LIN {X 0,Y 477.289,Z 363.649,A -85,B 0,C 180,E1 -7445.274,E2 -7445.274} C_VEL
LIN {X 0,Y 471.666,Z 382.664,A -85,B 0,C 180,E1 -7445.357,E2 -7445.357} C_VEL
LIN {X 0,Y 470.971,Z 388.509,A -85,B 0,C 180,E1 -7445.422,E2 -7445.422} C_VEL
LIN {X 0,Y 470.744,Z 411.297,A -85,B 0,C 180,E1 -7445.812,E2 -7445.812} C_VEL
LIN {X 0,Y 470.533,Z 424.379,A -85,B 0,C 180,E1 -7446.217,E2 -7446.217} C_VEL
LIN {X 0,Y 470.087,Z 436.738,A -85,B 0,C 180,E1 -7446.777,E2 -7446.777} C_VEL
LIN {X 0,Y 469.665,Z 447.889,A -85,B 0,C 180,E1 -7447.453,E2 -7447.453} C_VEL
LIN {X 0,Y 469.142,Z 459.604,A -85,B 0,C 180,E1 -7448.361,E2 -7448.361} C_VEL
LIN {X 0,Y 468.636,Z 469.87,A -85,B 0,C 180,E1 -7449.365,E2 -7449.365} C_VEL
LIN {X 0,Y 468.188,Z 479.141,A -85,B 0,C 180,E1 -7450.489,E2 -7450.489} C_VEL
LIN {X 0,Y 467.745,Z 486.733,A -85,B 0,C 180,E1 -7451.608,E2 -7451.608} C_VEL
LIN {X 0,Y 467.41,Z 494.144,A -85,B 0,C 180,E1 -7452.951,E2 -7452.951} C_VEL
LIN {X 0,Y 467.098,Z 500.27,A -85,B 0,C 180,E1 -7454.357,E2 -7454.357} C_VEL
LIN {X 0,Y 466.929,Z 504.578,A -85,B 0,C 180,E1 -7455.621,E2 -7455.621} C_VEL
LIN {X 0,Y 466.792,Z 508.016,A -85,B 0,C 180,E1 -7456.948,E2 -7456.948} C_VEL
LIN {X 0,Y 466.745,Z 510.263,A -85,B 0,C 180,E1 -7458.166,E2 -7458.166} C_VEL
LIN {X 0,Y 466.637,Z 511.87,A -85,B 0,C 180,E1 -7459.588,E2 -7459.588} C_VEL
LIN {X 0,Y 466.582,Z 512.309,A -85,B 0,C 180,E1 -7460.463,E2 -7460.463} C_VEL
LIN {X 0,Y 466.636,Z 512.343,A -85,B 0,C 180,E1 -7461.338,E2 -7461.338} C_VEL
LIN {X 0,Y 466.705,Z 511.259,A -85,B 0,C 180,E1 -7463.081,E2 -7463.081} C_VEL
LIN {X 0,Y 466.765,Z 510.083,A -85,B 0,C 180,E1 -7463.95,E2 -7463.95} C_VEL
LIN {X 0,Y 466.742,Z 508.508,A -85,B 0,C 180,E1 -7464.817,E2 -7464.817} C_VEL
LIN {X 0,Y 466.893,Z 505.337,A -85,B 0,C 180,E1 -7466.117,E2 -7466.117} C_VEL
LIN {X 0,Y 466.996,Z 501.127,A -85,B 0,C 180,E1 -7467.413,E2 -7467.413} C_VEL
LIN {X 0,Y 467.29,Z 494.749,A -85,B 0,C 180,E1 -7468.923,E2 -7468.923} C_VEL
LIN {X 0,Y 467.608,Z 487.78,A -85,B 0,C 180,E1 -7470.216,E2 -7470.216} C_VEL
LIN {X 0,Y 468.041,Z 479.089,A -85,B 0,C 180,E1 -7471.506,E2 -7471.506} C_VEL
LIN {X 0,Y 468.446,Z 469.254,A -85,B 0,C 180,E1 -7472.688,E2 -7472.688} C_VEL
LIN {X 0,Y 468.883,Z 459.22,A -85,B 0,C 180,E1 -7473.653,E2 -7473.653} C_VEL
LIN {X 0,Y 469.362,Z 448.098,A -85,B 0,C 180,E1 -7474.509,E2 -7474.509} C_VEL
LIN {X 0,Y 469.775,Z 437.576,A -85,B 0,C 180,E1 -7475.15,E2 -7475.15} C_VEL
LIN {X 0,Y 470.065,Z 424.945,A -85,B 0,C 180,E1 -7475.739,E2 -7475.739} C_VEL
LIN {X 0,Y 470.376,Z 412.214,A -85,B 0,C 180,E1 -7476.139,E2 -7476.139} C_VEL
LIN {X 0,Y 470.57,Z 394.34,A -85,B 0,C 180,E1 -7476.459,E2 -7476.459} C_VEL
LIN {X 0,Y 471.157,Z 315.376,A -85,B 0,C 180,E1 -7477.664,E2 -7477.664} C_VEL
LIN {X 0,Y 468.446,Z 301.546,A -85,B 0,C 180,E1 -7478,E2 -7478} C_VEL
LIN {X 0,Y 468.444,Z 292.876,A -85,B 0,C 180,E1 -7479.718,E2 -7479.718} C_VEL
LIN {X 0,Y 467.617,Z 287.24,A -85,B 0,C 180,E1 -7480.911,E2 -7480.911} C_VEL
LIN {X 0,Y 467.59,Z 287.239,A -85,B 0,C 180,E1 -7483.03,E2 -7483.03} C_VEL
LIN {X 0,Y 467.655,Z 287.227,A -85,B 0,C 180,E1 -7485.885,E2 -7485.885} C_VEL
LIN {X 0,Y 467.623,Z 287.232,A -85,B 0,C 180,E1 -7489.308,E2 -7489.308} C_VEL
LIN {X 0,Y 467.537,Z 287.242,A -85,B 0,C 180,E1 -7492.074,E2 -7492.074} C_VEL
LIN {X 0,Y 467.561,Z 287.247,A -85,B 0,C 180,E1 -7494.89,E2 -7494.89} C_VEL
LIN {X 0,Y 467.549,Z 287.24,A -85,B 0,C 180,E1 -7497.774,E2 -7497.774} C_VEL
LIN {X 0,Y 467.548,Z 287.248,A -85,B 0,C 180,E1 -7501.04,E2 -7501.04} C_VEL
LIN {X 0,Y 467.582,Z 287.236,A -85,B 0,C 180,E1 -7504.24,E2 -7504.24} C_VEL
LIN {X 0,Y 467.548,Z 287.248,A -85,B 0,C 180,E1 -7507.185,E2 -7507.185} C_VEL
LIN {X 0,Y 467.562,Z 287.238,A -85,B 0,C 180,E1 -7510.267,E2 -7510.267} C_VEL
LIN {X 0,Y 467.55,Z 287.242,A -85,B 0,C 180,E1 -7513.746,E2 -7513.746} C_VEL
LIN {X 0,Y 467.549,Z 287.24,A -85,B 0,C 180,E1 -7516.254,E2 -7516.254} C_VEL
LIN {X 0,Y 467.561,Z 287.242,A -85,B 0,C 180,E1 -7519.733,E2 -7519.733} C_VEL
LIN {X 0,Y 467.527,Z 287.243,A -85,B 0,C 180,E1 -7522.818,E2 -7522.818} C_VEL
LIN {X 0,Y 467.581,Z 287.241,A -85,B 0,C 180,E1 -7525.76,E2 -7525.76} C_VEL
LIN {X 0,Y 467.572,Z 287.238,A -85,B 0,C 180,E1 -7528.955,E2 -7528.955} C_VEL
LIN {X 0,Y 467.608,Z 287.233,A -85,B 0,C 180,E1 -7532.469,E2 -7532.469} C_VEL
LIN {X 0,Y 467.559,Z 287.24,A -85,B 0,C 180,E1 -7535.11,E2 -7535.11} C_VEL
LIN {X 0,Y 467.539,Z 287.248,A -85,B 0,C 180,E1 -7537.926,E2 -7537.926} C_VEL
LIN {X 0,Y 467.625,Z 287.231,A -85,B 0,C 180,E1 -7540.692,E2 -7540.692} C_VEL
LIN {X 0,Y 467.643,Z 287.232,A -85,B 0,C 180,E1 -7544.305,E2 -7544.305} C_VEL
LIN {X 0,Y 467.652,Z 287.233,A -85,B 0,C 180,E1 -7547.854,E2 -7547.854} C_VEL
LIN {X 0,Y 467.641,Z 287.229,A -85,B 0,C 180,E1 -7551.356,E2 -7551.356} C_VEL
LIN {X 0,Y 467.706,Z 287.226,A -85,B 0,C 180,E1 -7553.962,E2 -7553.962} C_VEL
LIN {X 0,Y 467.816,Z 287.207,A -85,B 0,C 180,E1 -7557.417,E2 -7557.417} C_VEL
LIN {X 0,Y 467.853,Z 287.207,A -85,B 0,C 180,E1 -7560,E2 -7560} C_VEL
LIN {X 0,Y 467.815,Z 287.212,A -85,B 0,C 180,E1 -7562.583,E2 -7562.583} C_VEL
LIN {X 0,Y 467.705,Z 287.224,A -85,B 0,C 180,E1 -7566.038,E2 -7566.038} C_VEL
LIN {X 0,Y 467.633,Z 287.236,A -85,B 0,C 180,E1 -7568.643,E2 -7568.643} C_VEL
LIN {X 0,Y 467.651,Z 287.23,A -85,B 0,C 180,E1 -7572.145,E2 -7572.145} C_VEL
LIN {X 0,Y 467.642,Z 287.228,A -85,B 0,C 180,E1 -7575.695,E2 -7575.695} C_VEL
LIN {X 0,Y 467.621,Z 287.232,A -85,B 0,C 180,E1 -7579.308,E2 -7579.308} C_VEL
LIN {X 0,Y 467.534,Z 287.242,A -85,B 0,C 180,E1 -7582.074,E2 -7582.074} C_VEL
LIN {X 0,Y 467.558,Z 287.247,A -85,B 0,C 180,E1 -7584.89,E2 -7584.89} C_VEL
LIN {X 0,Y 467.546,Z 287.24,A -85,B 0,C 180,E1 -7587.774,E2 -7587.774} C_VEL
LIN {X 0,Y 467.545,Z 287.248,A -85,B 0,C 180,E1 -7591.039,E2 -7591.039} C_VEL
LIN {X 0,Y 467.579,Z 287.236,A -85,B 0,C 180,E1 -7594.24,E2 -7594.24} C_VEL
LIN {X 0,Y 467.545,Z 287.248,A -85,B 0,C 180,E1 -7597.185,E2 -7597.185} C_VEL
LIN {X 0,Y 467.56,Z 287.238,A -85,B 0,C 180,E1 -7600.266,E2 -7600.266} C_VEL
LIN {X 0,Y 467.547,Z 287.242,A -85,B 0,C 180,E1 -7603.745,E2 -7603.745} C_VEL
LIN {X 0,Y 467.547,Z 287.24,A -85,B 0,C 180,E1 -7606.254,E2 -7606.254} C_VEL
LIN {X 0,Y 467.559,Z 287.242,A -85,B 0,C 180,E1 -7609.733,E2 -7609.733} C_VEL
LIN {X 0,Y 467.525,Z 287.244,A -85,B 0,C 180,E1 -7612.818,E2 -7612.818} C_VEL
LIN {X 0,Y 467.579,Z 287.241,A -85,B 0,C 180,E1 -7615.76,E2 -7615.76} C_VEL
LIN {X 0,Y 467.57,Z 287.238,A -85,B 0,C 180,E1 -7618.955,E2 -7618.955} C_VEL
LIN {X 0,Y 467.606,Z 287.237,A -85,B 0,C 180,E1 -7622.468,E2 -7622.468} C_VEL
LIN {X 0,Y 467.609,Z 287.435,A -85,B 0,C 180,E1 -7623.68,E2 -7623.68} C_VEL
LIN {X 0,Y 469.866,Z 299.396,A -85,B 0,C 180,E1 -7625.84,E2 -7625.84} C_VEL
LIN {X 0,Y 469.239,Z 315.502,A -85,B 0,C 180,E1 -7628.547,E2 -7628.547} C_VEL
LIN {X 0,Y 468.541,Z 334.109,A -85,B 0,C 180,E1 -7631.639,E2 -7631.639} C_VEL
LIN {X 0,Y 468.228,Z 342.74,A -85,B 0,C 180,E1 -7633.043,E2 -7633.043} C_VEL
LIN {X 0,Y 471.085,Z 362.265,A -85,B 0,C 180,E1 -7633.441,E2 -7633.441} C_VEL
LIN {X 0,Y 470.385,Z 451.256,A -85,B 0,C 180,E1 -7634.815,E2 -7634.815} C_VEL
LIN {X 0,Y 470.021,Z 464.565,A -85,B 0,C 180,E1 -7635.191,E2 -7635.191} C_VEL
LIN {X 0,Y 469.576,Z 476.765,A -85,B 0,C 180,E1 -7635.702,E2 -7635.702} C_VEL
LIN {X 0,Y 469.14,Z 488.265,A -85,B 0,C 180,E1 -7636.352,E2 -7636.352} C_VEL
LIN {X 0,Y 468.673,Z 499.421,A -85,B 0,C 180,E1 -7637.166,E2 -7637.166} C_VEL
LIN {X 0,Y 468.186,Z 510.665,A -85,B 0,C 180,E1 -7638.198,E2 -7638.198} C_VEL
LIN {X 0,Y 467.733,Z 519.319,A -85,B 0,C 180,E1 -7639.174,E2 -7639.174} C_VEL
LIN {X 0,Y 467.39,Z 527.297,A -85,B 0,C 180,E1 -7640.26,E2 -7640.26} C_VEL
LIN {X 0,Y 467.065,Z 535.094,A -85,B 0,C 180,E1 -7641.563,E2 -7641.563} C_VEL
LIN {X 0,Y 466.833,Z 542.26,A -85,B 0,C 180,E1 -7643.082,E2 -7643.082} C_VEL
LIN {X 0,Y 466.76,Z 547.034,A -85,B 0,C 180,E1 -7644.383,E2 -7644.383} C_VEL
LIN {X 0,Y 466.649,Z 550.678,A -85,B 0,C 180,E1 -7645.681,E2 -7645.681} C_VEL
LIN {X 0,Y 466.692,Z 552.565,A -85,B 0,C 180,E1 -7646.546,E2 -7646.546} C_VEL
LIN {X 0,Y 466.679,Z 553.979,A -85,B 0,C 180,E1 -7647.41,E2 -7647.41} C_VEL
LIN {X 0,Y 466.661,Z 554.984,A -85,B 0,C 180,E1 -7648.273,E2 -7648.273} C_VEL
LIN {X 0,Y 466.603,Z 555.821,A -85,B 0,C 180,E1 -7649.999,E2 -7649.999} C_VEL
LIN {X 0,Y 466.621,Z 555.612,A -85,B 0,C 180,E1 -7650.862,E2 -7650.862} C_VEL
LIN {X 0,Y 466.661,Z 555.006,A -85,B 0,C 180,E1 -7651.725,E2 -7651.725} C_VEL
LIN {X 0,Y 466.68,Z 554.011,A -85,B 0,C 180,E1 -7652.589,E2 -7652.589} C_VEL
LIN {X 0,Y 466.697,Z 552.616,A -85,B 0,C 180,E1 -7653.453,E2 -7653.453} C_VEL
LIN {X 0,Y 466.689,Z 549.674,A -85,B 0,C 180,E1 -7654.75,E2 -7654.75} C_VEL
LIN {X 0,Y 466.748,Z 545.7,A -85,B 0,C 180,E1 -7656.05,E2 -7656.05} C_VEL
LIN {X 0,Y 466.939,Z 539.601,A -85,B 0,C 180,E1 -7657.567,E2 -7657.567} C_VEL
LIN {X 0,Y 467.144,Z 532.934,A -85,B 0,C 180,E1 -7658.87,E2 -7658.87} C_VEL
LIN {X 0,Y 467.505,Z 524.674,A -85,B 0,C 180,E1 -7660.173,E2 -7660.173} C_VEL
LIN {X 0,Y 467.983,Z 516.238,A -85,B 0,C 180,E1 -7661.258,E2 -7661.258} C_VEL
LIN {X 0,Y 468.432,Z 506.296,A -85,B 0,C 180,E1 -7662.301,E2 -7662.301} C_VEL
LIN {X 0,Y 468.929,Z 495.565,A -85,B 0,C 180,E1 -7663.212,E2 -7663.212} C_VEL
LIN {X 0,Y 469.427,Z 484.35,A -85,B 0,C 180,E1 -7663.969,E2 -7663.969} C_VEL
LIN {X 0,Y 469.957,Z 471.778,A -85,B 0,C 180,E1 -7664.617,E2 -7664.617} C_VEL
LIN {X 0,Y 470.415,Z 458.336,A -85,B 0,C 180,E1 -7665.1,E2 -7665.1} C_VEL
LIN {X 0,Y 470.732,Z 445.029,A -85,B 0,C 180,E1 -7665.394,E2 -7665.394} C_VEL
LIN {X 0,Y 471.208,Z 361.262,A -85,B 0,C 180,E1 -7666.69,E2 -7666.69} C_VEL
LIN {X 0,Y 468.296,Z 342.345,A -85,B 0,C 180,E1 -7667.112,E2 -7667.112} C_VEL
LIN {X 0,Y 469.056,Z 324.114,A -85,B 0,C 180,E1 -7670.158,E2 -7670.158} C_VEL
LIN {X 0,Y 469.88,Z 305.296,A -85,B 0,C 180,E1 -7673.35,E2 -7673.35} C_VEL
LIN {X 0,Y 469.95,Z 299.136,A -85,B 0,C 180,E1 -7674.419,E2 -7674.419} C_VEL
LIN {X 0,Y 467.581,Z 287.244,A -85,B 0,C 180,E1 -7676.681,E2 -7676.681} C_VEL
LIN {X 0,Y 467.545,Z 287.251,A -85,B 0,C 180,E1 -7679.738,E2 -7679.738} C_VEL
LIN {X 0,Y 467.578,Z 287.247,A -85,B 0,C 180,E1 -7682.758,E2 -7682.758} C_VEL
LIN {X 0,Y 467.549,Z 287.247,A -85,B 0,C 180,E1 -7685.889,E2 -7685.889} C_VEL
LIN {X 0,Y 467.556,Z 287.24,A -85,B 0,C 180,E1 -7689.147,E2 -7689.147} C_VEL
LIN {X 0,Y 467.584,Z 287.243,A -85,B 0,C 180,E1 -7692.566,E2 -7692.566} C_VEL
LIN {X 0,Y 467.563,Z 287.241,A -85,B 0,C 180,E1 -7695.052,E2 -7695.052} C_VEL
LIN {X 0,Y 467.586,Z 287.237,A -85,B 0,C 180,E1 -7697.44,E2 -7697.44} C_VEL
LIN {X 0,Y 467.579,Z 287.24,A -85,B 0,C 180,E1 -7700.855,E2 -7700.855} C_VEL
LIN {X 0,Y 467.556,Z 287.244,A -85,B 0,C 180,E1 -7704.261,E2 -7704.261} C_VEL
LIN {X 0,Y 467.576,Z 287.237,A -85,B 0,C 180,E1 -7707.321,E2 -7707.321} C_VEL
LIN {X 0,Y 467.567,Z 287.244,A -85,B 0,C 180,E1 -7710.667,E2 -7710.667} C_VEL
LIN {X 0,Y 467.609,Z 287.234,A -85,B 0,C 180,E1 -7713.199,E2 -7713.199} C_VEL
LIN {X 0,Y 467.587,Z 287.237,A -85,B 0,C 180,E1 -7716.469,E2 -7716.469} C_VEL
LIN {X 0,Y 467.621,Z 287.227,A -85,B 0,C 180,E1 -7719.777,E2 -7719.777} C_VEL
LIN {X 0,Y 467.606,Z 287.239,A -85,B 0,C 180,E1 -7722.507,E2 -7722.507} C_VEL
LIN {X 0,Y 467.603,Z 287.237,A -85,B 0,C 180,E1 -7725.196,E2 -7725.196} C_VEL
LIN {X 0,Y 467.652,Z 287.224,A -85,B 0,C 180,E1 -7727.855,E2 -7727.855} C_VEL
LIN {X 0,Y 467.678,Z 287.223,A -85,B 0,C 180,E1 -7731.357,E2 -7731.357} C_VEL
LIN {X 0,Y 467.74,Z 287.217,A -85,B 0,C 180,E1 -7733.963,E2 -7733.963} C_VEL
LIN {X 0,Y 467.857,Z 287.204,A -85,B 0,C 180,E1 -7737.417,E2 -7737.417} C_VEL
LIN {X 0,Y 467.88,Z 287.197,A -85,B 0,C 180,E1 -7740,E2 -7740} C_VEL
LIN {X 0,Y 467.857,Z 287.205,A -85,B 0,C 180,E1 -7742.583,E2 -7742.583} C_VEL
LIN {X 0,Y 467.74,Z 287.215,A -85,B 0,C 180,E1 -7746.038,E2 -7746.038} C_VEL
LIN {X 0,Y 467.679,Z 287.227,A -85,B 0,C 180,E1 -7748.643,E2 -7748.643} C_VEL
LIN {X 0,Y 467.653,Z 287.227,A -85,B 0,C 180,E1 -7752.146,E2 -7752.146} C_VEL
LIN {X 0,Y 467.636,Z 287.231,A -85,B 0,C 180,E1 -7755.695,E2 -7755.695} C_VEL
LIN {X 0,Y 467.61,Z 287.235,A -85,B 0,C 180,E1 -7758.763,E2 -7758.763} C_VEL
LIN {X 0,Y 467.578,Z 287.241,A -85,B 0,C 180,E1 -7761.269,E2 -7761.269} C_VEL
LIN {X 0,Y 467.559,Z 287.24,A -85,B 0,C 180,E1 -7763.944,E2 -7763.944} C_VEL
LIN {X 0,Y 467.61,Z 287.236,A -85,B 0,C 180,E1 -7766.801,E2 -7766.801} C_VEL
LIN {X 0,Y 467.551,Z 287.242,A -85,B 0,C 180,E1 -7769.739,E2 -7769.739} C_VEL
LIN {X 0,Y 467.577,Z 287.236,A -85,B 0,C 180,E1 -7772.759,E2 -7772.759} C_VEL
LIN {X 0,Y 467.552,Z 287.241,A -85,B 0,C 180,E1 -7775.89,E2 -7775.89} C_VEL
LIN {X 0,Y 467.553,Z 287.243,A -85,B 0,C 180,E1 -7779.148,E2 -7779.148} C_VEL
LIN {X 0,Y 467.57,Z 287.244,A -85,B 0,C 180,E1 -7781.404,E2 -7781.404} C_VEL
LIN {X 0,Y 467.565,Z 287.244,A -85,B 0,C 180,E1 -7785.053,E2 -7785.053} C_VEL
LIN {X 0,Y 467.563,Z 287.241,A -85,B 0,C 180,E1 -7788.726,E2 -7788.726} C_VEL
LIN {X 0,Y 467.547,Z 287.244,A -85,B 0,C 180,E1 -7791.954,E2 -7791.954} C_VEL
LIN {X 0,Y 467.557,Z 287.241,A -85,B 0,C 180,E1 -7795.167,E2 -7795.167} C_VEL
LIN {X 0,Y 467.581,Z 287.241,A -85,B 0,C 180,E1 -7798.26,E2 -7798.26} C_VEL
LIN {X 0,Y 467.623,Z 287.382,A -85,B 0,C 180,E1 -7801.063,E2 -7801.063} C_VEL
LIN {X 0,Y 468.633,Z 293.31,A -85,B 0,C 180,E1 -7802.297,E2 -7802.297} C_VEL
LIN {X 0,Y 468.503,Z 301.675,A -85,B 0,C 180,E1 -7803.938,E2 -7803.938} C_VEL
LIN {X 0,Y 471.604,Z 316.633,A -85,B 0,C 180,E1 -7804.316,E2 -7804.316} C_VEL
LIN {X 0,Y 470.971,Z 388.509,A -85,B 0,C 180,E1 -7805.422,E2 -7805.422} C_VEL
LIN {X 0,Y 470.284,Z 394.35,A -85,B 0,C 180,E1 -7805.484,E2 -7805.484} C_VEL
LIN {X 0,Y 464.61,Z 413.288,A -85,B 0,C 180,E1 -7805.626,E2 -7805.626} C_VEL
LIN {X 0,Y 463.861,Z 419.027,A -85,B 0,C 180,E1 -7805.769,E2 -7805.769} C_VEL
LIN {X 0,Y 463.473,Z 431.291,A -85,B 0,C 180,E1 -7806.248,E2 -7806.248} C_VEL
LIN {X 0,Y 463.027,Z 442.905,A -85,B 0,C 180,E1 -7806.876,E2 -7806.876} C_VEL
LIN {X 0,Y 462.563,Z 454.315,A -85,B 0,C 180,E1 -7807.677,E2 -7807.677} C_VEL
LIN {X 0,Y 461.983,Z 464.672,A -85,B 0,C 180,E1 -7808.587,E2 -7808.587} C_VEL
LIN {X 0,Y 461.467,Z 475.022,A -85,B 0,C 180,E1 -7809.729,E2 -7809.729} C_VEL
LIN {X 0,Y 460.931,Z 484.097,A -85,B 0,C 180,E1 -7810.97,E2 -7810.97} C_VEL
LIN {X 0,Y 460.53,Z 491.564,A -85,B 0,C 180,E1 -7812.23,E2 -7812.23} C_VEL
LIN {X 0,Y 460.209,Z 498.027,A -85,B 0,C 180,E1 -7813.59,E2 -7813.59} C_VEL
LIN {X 0,Y 459.949,Z 503.109,A -85,B 0,C 180,E1 -7814.945,E2 -7814.945} C_VEL
LIN {X 0,Y 459.764,Z 507.01,A -85,B 0,C 180,E1 -7816.295,E2 -7816.295} C_VEL
LIN {X 0,Y 459.658,Z 510.607,A -85,B 0,C 180,E1 -7818.111,E2 -7818.111} C_VEL
LIN {X 0,Y 459.576,Z 512.093,A -85,B 0,C 180,E1 -7819.426,E2 -7819.426} C_VEL
LIN {X 0,Y 459.495,Z 512.616,A -85,B 0,C 180,E1 -7820.315,E2 -7820.315} C_VEL
LIN {X 0,Y 459.53,Z 512.697,A -85,B 0,C 180,E1 -7821.203,E2 -7821.203} C_VEL
LIN {X 0,Y 459.618,Z 511.7,A -85,B 0,C 180,E1 -7822.974,E2 -7822.974} C_VEL
LIN {X 0,Y 459.669,Z 510.609,A -85,B 0,C 180,E1 -7823.857,E2 -7823.857} C_VEL
LIN {X 0,Y 459.673,Z 509.077,A -85,B 0,C 180,E1 -7824.737,E2 -7824.737} C_VEL
LIN {X 0,Y 459.809,Z 505.999,A -85,B 0,C 180,E1 -7826.057,E2 -7826.057} C_VEL
LIN {X 0,Y 459.931,Z 501.886,A -85,B 0,C 180,E1 -7827.373,E2 -7827.373} C_VEL
LIN {X 0,Y 460.195,Z 495.616,A -85,B 0,C 180,E1 -7828.907,E2 -7828.907} C_VEL
LIN {X 0,Y 460.555,Z 488.798,A -85,B 0,C 180,E1 -7830.219,E2 -7830.219} C_VEL
LIN {X 0,Y 460.99,Z 480.276,A -85,B 0,C 180,E1 -7831.529,E2 -7831.529} C_VEL
LIN {X 0,Y 461.361,Z 471.57,A -85,B 0,C 180,E1 -7832.62,E2 -7832.62} C_VEL
LIN {X 0,Y 461.805,Z 462.02,A -85,B 0,C 180,E1 -7833.6,E2 -7833.6} C_VEL
LIN {X 0,Y 462.315,Z 451.567,A -85,B 0,C 180,E1 -7834.469,E2 -7834.469} C_VEL
LIN {X 0,Y 462.867,Z 439.939,A -85,B 0,C 180,E1 -7835.228,E2 -7835.228} C_VEL
LIN {X 0,Y 463.126,Z 429.23,A -85,B 0,C 180,E1 -7835.771,E2 -7835.771} C_VEL
LIN {X 0,Y 463.387,Z 416.669,A -85,B 0,C 180,E1 -7836.231,E2 -7836.231} C_VEL
LIN {X 0,Y 463.71,Z 403.619,A -85,B 0,C 180,E1 -7836.527,E2 -7836.527} C_VEL
LIN {X 0,Y 464.307,Z 316.209,A -85,B 0,C 180,E1 -7837.884,E2 -7837.884} C_VEL
LIN {X 0,Y 461.518,Z 301.915,A -85,B 0,C 180,E1 -7838.22,E2 -7838.22} C_VEL
LIN {X 0,Y 461.439,Z 293.689,A -85,B 0,C 180,E1 -7839.867,E2 -7839.867} C_VEL
LIN {X 0,Y 460.559,Z 288.118,A -85,B 0,C 180,E1 -7841.053,E2 -7841.053} C_VEL
LIN {X 0,Y 460.545,Z 288.115,A -85,B 0,C 180,E1 -7843.233,E2 -7843.233} C_VEL
LIN {X 0,Y 460.607,Z 288.105,A -85,B 0,C 180,E1 -7845.998,E2 -7845.998} C_VEL
LIN {X 0,Y 460.57,Z 288.109,A -85,B 0,C 180,E1 -7849.616,E2 -7849.616} C_VEL
LIN {X 0,Y 460.513,Z 288.12,A -85,B 0,C 180,E1 -7852.429,E2 -7852.429} C_VEL
LIN {X 0,Y 460.538,Z 288.113,A -85,B 0,C 180,E1 -7855.793,E2 -7855.793} C_VEL
LIN {X 0,Y 460.521,Z 288.12,A -85,B 0,C 180,E1 -7859.233,E2 -7859.233} C_VEL
LIN {X 0,Y 460.523,Z 288.116,A -85,B 0,C 180,E1 -7862.286,E2 -7862.286} C_VEL
LIN {X 0,Y 460.512,Z 288.12,A -85,B 0,C 180,E1 -7865.446,E2 -7865.446} C_VEL
LIN {X 0,Y 460.509,Z 288.121,A -85,B 0,C 180,E1 -7868.891,E2 -7868.891} C_VEL
LIN {X 0,Y 460.507,Z 288.121,A -85,B 0,C 180,E1 -7871.598,E2 -7871.598} C_VEL
LIN {X 0,Y 460.516,Z 288.117,A -85,B 0,C 180,E1 -7874.589,E2 -7874.589} C_VEL
LIN {X 0,Y 460.48,Z 288.123,A -85,B 0,C 180,E1 -7877.813,E2 -7877.813} C_VEL
LIN {X 0,Y 460.515,Z 288.117,A -85,B 0,C 180,E1 -7880.135,E2 -7880.135} C_VEL
LIN {X 0,Y 460.47,Z 288.13,A -85,B 0,C 180,E1 -7883.469,E2 -7883.469} C_VEL
LIN {X 0,Y 460.521,Z 288.115,A -85,B 0,C 180,E1 -7886.674,E2 -7886.674} C_VEL
LIN {X 0,Y 460.512,Z 288.123,A -85,B 0,C 180,E1 -7889.76,E2 -7889.76} C_VEL
LIN {X 0,Y 460.532,Z 288.114,A -85,B 0,C 180,E1 -7892.753,E2 -7892.753} C_VEL
LIN {X 0,Y 460.52,Z 288.123,A -85,B 0,C 180,E1 -7895.666,E2 -7895.666} C_VEL
LIN {X 0,Y 460.527,Z 288.115,A -85,B 0,C 180,E1 -7898.578,E2 -7898.578} C_VEL
LIN {X 0,Y 460.589,Z 288.108,A -85,B 0,C 180,E1 -7901.311,E2 -7901.311} C_VEL
LIN {X 0,Y 460.61,Z 288.111,A -85,B 0,C 180,E1 -7904.059,E2 -7904.059} C_VEL
LIN {X 0,Y 460.608,Z 288.108,A -85,B 0,C 180,E1 -7907.666,E2 -7907.666} C_VEL
LIN {X 0,Y 460.595,Z 288.106,A -85,B 0,C 180,E1 -7911.223,E2 -7911.223} C_VEL
LIN {X 0,Y 460.673,Z 288.101,A -85,B 0,C 180,E1 -7913.869,E2 -7913.869} C_VEL
LIN {X 0,Y 460.76,Z 288.086,A -85,B 0,C 180,E1 -7917.377,E2 -7917.377} C_VEL
LIN {X 0,Y 460.822,Z 288.082,A -85,B 0,C 180,E1 -7920,E2 -7920} C_VEL
LIN {X 0,Y 460.759,Z 288.09,A -85,B 0,C 180,E1 -7922.623,E2 -7922.623} C_VEL
LIN {X 0,Y 460.671,Z 288.101,A -85,B 0,C 180,E1 -7926.13,E2 -7926.13} C_VEL
LIN {X 0,Y 460.588,Z 288.111,A -85,B 0,C 180,E1 -7928.777,E2 -7928.777} C_VEL
LIN {X 0,Y 460.601,Z 288.112,A -85,B 0,C 180,E1 -7932.435,E2 -7932.435} C_VEL
LIN {X 0,Y 460.583,Z 288.109,A -85,B 0,C 180,E1 -7935.988,E2 -7935.988} C_VEL
LIN {X 0,Y 460.568,Z 288.109,A -85,B 0,C 180,E1 -7939.615,E2 -7939.615} C_VEL
LIN {X 0,Y 460.511,Z 288.12,A -85,B 0,C 180,E1 -7942.429,E2 -7942.429} C_VEL
LIN {X 0,Y 460.535,Z 288.113,A -85,B 0,C 180,E1 -7945.792,E2 -7945.792} C_VEL
LIN {X 0,Y 460.519,Z 288.12,A -85,B 0,C 180,E1 -7949.232,E2 -7949.232} C_VEL
LIN {X 0,Y 460.52,Z 288.116,A -85,B 0,C 180,E1 -7952.285,E2 -7952.285} C_VEL
LIN {X 0,Y 460.509,Z 288.12,A -85,B 0,C 180,E1 -7955.446,E2 -7955.446} C_VEL
LIN {X 0,Y 460.506,Z 288.122,A -85,B 0,C 180,E1 -7958.891,E2 -7958.891} C_VEL
LIN {X 0,Y 460.504,Z 288.121,A -85,B 0,C 180,E1 -7961.598,E2 -7961.598} C_VEL
LIN {X 0,Y 460.514,Z 288.117,A -85,B 0,C 180,E1 -7964.589,E2 -7964.589} C_VEL
LIN {X 0,Y 460.477,Z 288.123,A -85,B 0,C 180,E1 -7967.813,E2 -7967.813} C_VEL
LIN {X 0,Y 460.513,Z 288.117,A -85,B 0,C 180,E1 -7970.135,E2 -7970.135} C_VEL
LIN {X 0,Y 460.468,Z 288.131,A -85,B 0,C 180,E1 -7973.469,E2 -7973.469} C_VEL
LIN {X 0,Y 460.519,Z 288.116,A -85,B 0,C 180,E1 -7976.674,E2 -7976.674} C_VEL
LIN {X 0,Y 460.51,Z 288.125,A -85,B 0,C 180,E1 -7979.759,E2 -7979.759} C_VEL
LIN {X 0,Y 460.535,Z 288.118,A -85,B 0,C 180,E1 -7982.753,E2 -7982.753} C_VEL
LIN {X 0,Y 460.571,Z 288.272,A -85,B 0,C 180,E1 -7983.491,E2 -7983.491} C_VEL
LIN {X 0,Y 462.891,Z 300.865,A -85,B 0,C 180,E1 -7985.799,E2 -7985.799} C_VEL
LIN {X 0,Y 462.293,Z 315.517,A -85,B 0,C 180,E1 -7988.297,E2 -7988.297} C_VEL
LIN {X 0,Y 461.588,Z 333.626,A -85,B 0,C 180,E1 -7991.352,E2 -7991.352} C_VEL
LIN {X 0,Y 461.196,Z 342.269,A -85,B 0,C 180,E1 -7992.799,E2 -7992.799} C_VEL
LIN {X 0,Y 464.22,Z 362.818,A -85,B 0,C 180,E1 -7993.226,E2 -7993.226} C_VEL
LIN {X 0,Y 463.489,Z 451.172,A -85,B 0,C 180,E1 -7994.611,E2 -7994.611} C_VEL
LIN {X 0,Y 463.1,Z 464.404,A -85,B 0,C 180,E1 -7994.992,E2 -7994.992} C_VEL
LIN {X 0,Y 462.639,Z 477.138,A -85,B 0,C 180,E1 -7995.539,E2 -7995.539} C_VEL
LIN {X 0,Y 462.137,Z 489.246,A -85,B 0,C 180,E1 -7996.253,E2 -7996.253} C_VEL
LIN {X 0,Y 461.625,Z 501.082,A -85,B 0,C 180,E1 -7997.158,E2 -7997.158} C_VEL
LIN {X 0,Y 461.143,Z 511.221,A -85,B 0,C 180,E1 -7998.126,E2 -7998.126} C_VEL
LIN {X 0,Y 460.618,Z 520.563,A -85,B 0,C 180,E1 -7999.227,E2 -7999.227} C_VEL
LIN {X 0,Y 460.198,Z 529.627,A -85,B 0,C 180,E1 -8000.55,E2 -8000.55} C_VEL
LIN {X 0,Y 459.927,Z 536.929,A -85,B 0,C 180,E1 -8001.874,E2 -8001.874} C_VEL
LIN {X 0,Y 459.738,Z 543.055,A -85,B 0,C 180,E1 -8003.272,E2 -8003.272} C_VEL
LIN {X 0,Y 459.667,Z 547.989,A -85,B 0,C 180,E1 -8004.736,E2 -8004.736} C_VEL
LIN {X 0,Y 459.566,Z 550.31,A -85,B 0,C 180,E1 -8005.614,E2 -8005.614} C_VEL
LIN {X 0,Y 459.589,Z 552.204,A -85,B 0,C 180,E1 -8006.493,E2 -8006.493} C_VEL
LIN {X 0,Y 459.6,Z 553.629,A -85,B 0,C 180,E1 -8007.37,E2 -8007.37} C_VEL
LIN {X 0,Y 459.554,Z 555.26,A -85,B 0,C 180,E1 -8009.123,E2 -8009.123} C_VEL
LIN {X 0,Y 459.535,Z 555.49,A -85,B 0,C 180,E1 -8009.999,E2 -8009.999} C_VEL
LIN {X 0,Y 459.554,Z 555.291,A -85,B 0,C 180,E1 -8010.876,E2 -8010.876} C_VEL
LIN {X 0,Y 459.601,Z 553.7,A -85,B 0,C 180,E1 -8012.629,E2 -8012.629} C_VEL
LIN {X 0,Y 459.593,Z 552.311,A -85,B 0,C 180,E1 -8013.506,E2 -8013.506} C_VEL
LIN {X 0,Y 459.616,Z 549.382,A -85,B 0,C 180,E1 -8014.824,E2 -8014.824} C_VEL
LIN {X 0,Y 459.713,Z 544.406,A -85,B 0,C 180,E1 -8016.43,E2 -8016.43} C_VEL
LIN {X 0,Y 459.884,Z 538.332,A -85,B 0,C 180,E1 -8017.905,E2 -8017.905} C_VEL
LIN {X 0,Y 460.165,Z 531.464,A -85,B 0,C 180,E1 -8019.227,E2 -8019.227} C_VEL
LIN {X 0,Y 460.547,Z 522.916,A -85,B 0,C 180,E1 -8020.551,E2 -8020.551} C_VEL
LIN {X 0,Y 461.054,Z 514.147,A -85,B 0,C 180,E1 -8021.652,E2 -8021.652} C_VEL
LIN {X 0,Y 461.585,Z 503.421,A -85,B 0,C 180,E1 -8022.749,E2 -8022.749} C_VEL
LIN {X 0,Y 462.145,Z 492.629,A -85,B 0,C 180,E1 -8023.633,E2 -8023.633} C_VEL
LIN {X 0,Y 462.71,Z 480.6,A -85,B 0,C 180,E1 -8024.401,E2 -8024.401} C_VEL
LIN {X 0,Y 463.229,Z 468.077,A -85,B 0,C 180,E1 -8025.002,E2 -8025.002} C_VEL
LIN {X 0,Y 463.705,Z 454.933,A -85,B 0,C 180,E1 -8025.437,E2 -8025.437} C_VEL
LIN {X 0,Y 463.967,Z 439.075,A -85,B 0,C 180,E1 -8025.737,E2 -8025.737} C_VEL
LIN {X 0,Y 464.45,Z 361.891,A -85,B 0,C 180,E1 -8026.949,E2 -8026.949} C_VEL
LIN {X 0,Y 461.357,Z 342.044,A -85,B 0,C 180,E1 -8027.397,E2 -8027.397} C_VEL
LIN {X 0,Y 462.098,Z 325.285,A -85,B 0,C 180,E1 -8030.242,E2 -8030.242} C_VEL
LIN {X 0,Y 462.963,Z 306.484,A -85,B 0,C 180,E1 -8033.483,E2 -8033.483} C_VEL
LIN {X 0,Y 463.115,Z 301.139,A -85,B 0,C 180,E1 -8034.421,E2 -8034.421} C_VEL
LIN {X 0,Y 460.984,Z 290.307,A -85,B 0,C 180,E1 -8036.483,E2 -8036.483} C_VEL
LIN {X 0,Y 460.553,Z 288.12,A -85,B 0,C 180,E1 -8036.938,E2 -8036.938} C_VEL
LIN {X 0,Y 460.505,Z 288.13,A -85,B 0,C 180,E1 -8040.24,E2 -8040.24} C_VEL
LIN {X 0,Y 460.518,Z 288.123,A -85,B 0,C 180,E1 -8043.325,E2 -8043.325} C_VEL
LIN {X 0,Y 460.47,Z 288.13,A -85,B 0,C 180,E1 -8046.529,E2 -8046.529} C_VEL
LIN {X 0,Y 460.522,Z 288.118,A -85,B 0,C 180,E1 -8049.863,E2 -8049.863} C_VEL
LIN {X 0,Y 460.51,Z 288.121,A -85,B 0,C 180,E1 -8052.9,E2 -8052.9} C_VEL
LIN {X 0,Y 460.506,Z 288.12,A -85,B 0,C 180,E1 -8055.83,E2 -8055.83} C_VEL
LIN {X 0,Y 460.528,Z 288.116,A -85,B 0,C 180,E1 -8058.988,E2 -8058.988} C_VEL
LIN {X 0,Y 460.523,Z 288.115,A -85,B 0,C 180,E1 -8061.267,E2 -8061.267} C_VEL
LIN {X 0,Y 460.505,Z 288.123,A -85,B 0,C 180,E1 -8064.554,E2 -8064.554} C_VEL
LIN {X 0,Y 460.526,Z 288.114,A -85,B 0,C 180,E1 -8067.715,E2 -8067.715} C_VEL
LIN {X 0,Y 460.536,Z 288.118,A -85,B 0,C 180,E1 -8070.769,E2 -8070.769} C_VEL
LIN {X 0,Y 460.552,Z 288.111,A -85,B 0,C 180,E1 -8073.734,E2 -8073.734} C_VEL
LIN {X 0,Y 460.541,Z 288.117,A -85,B 0,C 180,E1 -8076.624,E2 -8076.624} C_VEL
LIN {X 0,Y 460.548,Z 288.109,A -85,B 0,C 180,E1 -8079.453,E2 -8079.453} C_VEL
LIN {X 0,Y 460.556,Z 288.114,A -85,B 0,C 180,E1 -8082.23,E2 -8082.23} C_VEL
LIN {X 0,Y 460.562,Z 288.117,A -85,B 0,C 180,E1 -8084.965,E2 -8084.965} C_VEL
LIN {X 0,Y 460.608,Z 288.106,A -85,B 0,C 180,E1 -8088.559,E2 -8088.559} C_VEL
LIN {X 0,Y 460.692,Z 288.092,A -85,B 0,C 180,E1 -8092.109,E2 -8092.109} C_VEL
LIN {X 0,Y 460.694,Z 288.101,A -85,B 0,C 180,E1 -8094.748,E2 -8094.748} C_VEL
LIN {X 0,Y 460.822,Z 288.081,A -85,B 0,C 180,E1 -8097.378,E2 -8097.378} C_VEL
LIN {X 0,Y 460.851,Z 288.073,A -85,B 0,C 180,E1 -8100,E2 -8100} C_VEL
LIN {X 0,Y 460.821,Z 288.082,A -85,B 0,C 180,E1 -8102.623,E2 -8102.623} C_VEL
LIN {X 0,Y 460.706,Z 288.092,A -85,B 0,C 180,E1 -8106.13,E2 -8106.13} C_VEL
LIN {X 0,Y 460.626,Z 288.107,A -85,B 0,C 180,E1 -8108.776,E2 -8108.776} C_VEL
LIN {X 0,Y 460.61,Z 288.106,A -85,B 0,C 180,E1 -8112.445,E2 -8112.445} C_VEL
LIN {X 0,Y 460.597,Z 288.106,A -85,B 0,C 180,E1 -8115.998,E2 -8115.998} C_VEL
LIN {X 0,Y 460.565,Z 288.113,A -85,B 0,C 180,E1 -8119.616,E2 -8119.616} C_VEL
LIN {X 0,Y 460.508,Z 288.117,A -85,B 0,C 180,E1 -8122.429,E2 -8122.429} C_VEL
LIN {X 0,Y 460.55,Z 288.113,A -85,B 0,C 180,E1 -8125.799,E2 -8125.799} C_VEL
LIN {X 0,Y 460.549,Z 288.112,A -85,B 0,C 180,E1 -8128.234,E2 -8128.234} C_VEL
LIN {X 0,Y 460.518,Z 288.121,A -85,B 0,C 180,E1 -8131.283,E2 -8131.283} C_VEL
LIN {X 0,Y 460.522,Z 288.116,A -85,B 0,C 180,E1 -8134.505,E2 -8134.505} C_VEL
LIN {X 0,Y 460.499,Z 288.12,A -85,B 0,C 180,E1 -8137.624,E2 -8137.624} C_VEL
LIN {X 0,Y 460.525,Z 288.119,A -85,B 0,C 180,E1 -8141.013,E2 -8141.013} C_VEL
LIN {X 0,Y 460.511,Z 288.119,A -85,B 0,C 180,E1 -8144.59,E2 -8144.59} C_VEL
LIN {X 0,Y 460.49,Z 288.125,A -85,B 0,C 180,E1 -8147.816,E2 -8147.816} C_VEL
LIN {X 0,Y 460.51,Z 288.12,A -85,B 0,C 180,E1 -8150.136,E2 -8150.136} C_VEL
LIN {X 0,Y 460.466,Z 288.131,A -85,B 0,C 180,E1 -8153.47,E2 -8153.47} C_VEL
LIN {X 0,Y 460.52,Z 288.118,A -85,B 0,C 180,E1 -8156.675,E2 -8156.675} C_VEL
LIN {X 0,Y 460.507,Z 288.126,A -85,B 0,C 180,E1 -8159.76,E2 -8159.76} C_VEL
LIN {X 0,Y 460.565,Z 288.233,A -85,B 0,C 180,E1 -8160.834,E2 -8160.834} C_VEL
LIN {X 0,Y 461.651,Z 293.738,A -85,B 0,C 180,E1 -8162.004,E2 -8162.004} C_VEL
LIN {X 0,Y 461.63,Z 301.982,A -85,B 0,C 180,E1 -8163.647,E2 -8163.647} C_VEL
LIN {X 0,Y 464.904,Z 317.609,A -85,B 0,C 180,E1 -8164.052,E2 -8164.052} C_VEL
LIN {X 0,Y 463.969,Z 409.712,A -85,B 0,C 180,E1 -8165.511,E2 -8165.511} C_VEL
LIN {X 0,Y 463.861,Z 419.027,A -85,B 0,C 180,E1 -8165.769,E2 -8165.769} C_VEL
LIN {X 0,Y 463.028,Z 424.731,A -85,B 0,C 180,E1 -8165.935,E2 -8165.935} C_VEL
LIN {X 0,Y 459.997,Z 433.884,A -85,B 0,C 180,E1 -8166.227,E2 -8166.227} C_VEL
LIN {X 0,Y 456.921,Z 442.733,A -85,B 0,C 180,E1 -8166.62,E2 -8166.62} C_VEL
LIN {X 0,Y 456.019,Z 447.95,A -85,B 0,C 180,E1 -8166.943,E2 -8166.943} C_VEL
LIN {X 0,Y 455.474,Z 458.779,A -85,B 0,C 180,E1 -8167.791,E2 -8167.791} C_VEL
LIN {X 0,Y 454.851,Z 469.403,A -85,B 0,C 180,E1 -8168.828,E2 -8168.828} C_VEL
LIN {X 0,Y 454.393,Z 478.051,A -85,B 0,C 180,E1 -8169.872,E2 -8169.872} C_VEL
LIN {X 0,Y 453.894,Z 485.943,A -85,B 0,C 180,E1 -8171.025,E2 -8171.025} C_VEL
LIN {X 0,Y 453.428,Z 493.605,A -85,B 0,C 180,E1 -8172.408,E2 -8172.408} C_VEL
LIN {X 0,Y 453.112,Z 499.714,A -85,B 0,C 180,E1 -8173.789,E2 -8173.789} C_VEL
LIN {X 0,Y 452.874,Z 504.504,A -85,B 0,C 180,E1 -8175.164,E2 -8175.164} C_VEL
LIN {X 0,Y 452.684,Z 508.133,A -85,B 0,C 180,E1 -8176.534,E2 -8176.534} C_VEL
LIN {X 0,Y 452.572,Z 510.956,A -85,B 0,C 180,E1 -8178.053,E2 -8178.053} C_VEL
LIN {X 0,Y 452.505,Z 512.318,A -85,B 0,C 180,E1 -8179.259,E2 -8179.259} C_VEL
LIN {X 0,Y 452.412,Z 512.895,A -85,B 0,C 180,E1 -8180.162,E2 -8180.162} C_VEL
LIN {X 0,Y 452.44,Z 513.05,A -85,B 0,C 180,E1 -8181.064,E2 -8181.064} C_VEL
LIN {X 0,Y 452.534,Z 512.136,A -85,B 0,C 180,E1 -8182.864,E2 -8182.864} C_VEL
LIN {X 0,Y 452.587,Z 511.103,A -85,B 0,C 180,E1 -8183.76,E2 -8183.76} C_VEL
LIN {X 0,Y 452.604,Z 509.64,A -85,B 0,C 180,E1 -8184.655,E2 -8184.655} C_VEL
LIN {X 0,Y 452.727,Z 506.653,A -85,B 0,C 180,E1 -8185.995,E2 -8185.995} C_VEL
LIN {X 0,Y 452.867,Z 502.634,A -85,B 0,C 180,E1 -8187.332,E2 -8187.332} C_VEL
LIN {X 0,Y 453.109,Z 496.47,A -85,B 0,C 180,E1 -8188.89,E2 -8188.89} C_VEL
LIN {X 0,Y 453.503,Z 489.761,A -85,B 0,C 180,E1 -8190.223,E2 -8190.223} C_VEL
LIN {X 0,Y 453.941,Z 481.441,A -85,B 0,C 180,E1 -8191.553,E2 -8191.553} C_VEL
LIN {X 0,Y 454.338,Z 472.895,A -85,B 0,C 180,E1 -8192.66,E2 -8192.66} C_VEL
LIN {X 0,Y 454.849,Z 462.385,A -85,B 0,C 180,E1 -8193.766,E2 -8193.766} C_VEL
LIN {X 0,Y 455.367,Z 451.94,A -85,B 0,C 180,E1 -8194.648,E2 -8194.648} C_VEL
LIN {X 0,Y 455.95,Z 440.323,A -85,B 0,C 180,E1 -8195.418,E2 -8195.418} C_VEL
LIN {X 0,Y 456.224,Z 429.627,A -85,B 0,C 180,E1 -8195.969,E2 -8195.969} C_VEL
LIN {X 0,Y 456.503,Z 417.085,A -85,B 0,C 180,E1 -8196.437,E2 -8196.437} C_VEL
LIN {X 0,Y 456.833,Z 404.094,A -85,B 0,C 180,E1 -8196.737,E2 -8196.737} C_VEL
LIN {X 0,Y 457.559,Z 317.635,A -85,B 0,C 180,E1 -8198.096,E2 -8198.096} C_VEL
LIN {X 0,Y 454.587,Z 302.169,A -85,B 0,C 180,E1 -8198.469,E2 -8198.469} C_VEL
LIN {X 0,Y 454.425,Z 294.515,A -85,B 0,C 180,E1 -8200.02,E2 -8200.02} C_VEL
LIN {X 0,Y 453.54,Z 288.992,A -85,B 0,C 180,E1 -8201.226,E2 -8201.226} C_VEL
LIN {X 0,Y 453.507,Z 288.991,A -85,B 0,C 180,E1 -8203.442,E2 -8203.442} C_VEL
LIN {X 0,Y 453.55,Z 288.986,A -85,B 0,C 180,E1 -8206.196,E2 -8206.196} C_VEL
LIN {X 0,Y 453.523,Z 288.991,A -85,B 0,C 180,E1 -8209.039,E2 -8209.039} C_VEL
LIN {X 0,Y 453.482,Z 288.992,A -85,B 0,C 180,E1 -8211.836,E2 -8211.836} C_VEL
LIN {X 0,Y 453.491,Z 288.998,A -85,B 0,C 180,E1 -8214.736,E2 -8214.736} C_VEL
LIN {X 0,Y 453.467,Z 288.994,A -85,B 0,C 180,E1 -8217.943,E2 -8217.943} C_VEL
LIN {X 0,Y 453.46,Z 289,A -85,B 0,C 180,E1 -8220.761,E2 -8220.761} C_VEL
LIN {X 0,Y 453.472,Z 288.994,A -85,B 0,C 180,E1 -8223.914,E2 -8223.914} C_VEL
LIN {X 0,Y 453.455,Z 289.004,A -85,B 0,C 180,E1 -8227.19,E2 -8227.19} C_VEL
LIN {X 0,Y 453.475,Z 288.994,A -85,B 0,C 180,E1 -8230.612,E2 -8230.612} C_VEL
LIN {X 0,Y 453.486,Z 288.992,A -85,B 0,C 180,E1 -8234.528,E2 -8234.528} C_VEL
LIN {X 0,Y 453.441,Z 288.998,A -85,B 0,C 180,E1 -8238.071,E2 -8238.071} C_VEL
LIN {X 0,Y 453.447,Z 288.998,A -85,B 0,C 180,E1 -8240.802,E2 -8240.802} C_VEL
LIN {X 0,Y 453.453,Z 288.999,A -85,B 0,C 180,E1 -8243.916,E2 -8243.916} C_VEL
LIN {X 0,Y 453.48,Z 288.995,A -85,B 0,C 180,E1 -8247.15,E2 -8247.15} C_VEL
LIN {X 0,Y 453.471,Z 288.995,A -85,B 0,C 180,E1 -8250.268,E2 -8250.268} C_VEL
LIN {X 0,Y 453.464,Z 288.997,A -85,B 0,C 180,E1 -8253.291,E2 -8253.291} C_VEL
LIN {X 0,Y 453.497,Z 288.993,A -85,B 0,C 180,E1 -8256.238,E2 -8256.238} C_VEL
LIN {X 0,Y 453.487,Z 288.992,A -85,B 0,C 180,E1 -8259.117,E2 -8259.117} C_VEL
LIN {X 0,Y 453.503,Z 288.998,A -85,B 0,C 180,E1 -8261.944,E2 -8261.944} C_VEL
LIN {X 0,Y 453.542,Z 288.985,A -85,B 0,C 180,E1 -8264.726,E2 -8264.726} C_VEL
LIN {X 0,Y 453.549,Z 288.988,A -85,B 0,C 180,E1 -8268.378,E2 -8268.378} C_VEL
LIN {X 0,Y 453.565,Z 288.982,A -85,B 0,C 180,E1 -8271.086,E2 -8271.086} C_VEL
LIN {X 0,Y 453.64,Z 288.976,A -85,B 0,C 180,E1 -8273.774,E2 -8273.774} C_VEL
LIN {X 0,Y 453.707,Z 288.964,A -85,B 0,C 180,E1 -8277.336,E2 -8277.336} C_VEL
LIN {X 0,Y 453.771,Z 288.961,A -85,B 0,C 180,E1 -8280,E2 -8280} C_VEL
LIN {X 0,Y 453.705,Z 288.968,A -85,B 0,C 180,E1 -8282.663,E2 -8282.663} C_VEL
LIN {X 0,Y 453.639,Z 288.978,A -85,B 0,C 180,E1 -8286.226,E2 -8286.226} C_VEL
LIN {X 0,Y 453.558,Z 288.986,A -85,B 0,C 180,E1 -8288.914,E2 -8288.914} C_VEL
LIN {X 0,Y 453.568,Z 288.99,A -85,B 0,C 180,E1 -8292.529,E2 -8292.529} C_VEL
LIN {X 0,Y 453.541,Z 288.987,A -85,B 0,C 180,E1 -8296.196,E2 -8296.196} C_VEL
LIN {X 0,Y 453.521,Z 288.991,A -85,B 0,C 180,E1 -8299.039,E2 -8299.039} C_VEL
LIN {X 0,Y 453.479,Z 288.992,A -85,B 0,C 180,E1 -8301.836,E2 -8301.836} C_VEL
LIN {X 0,Y 453.489,Z 288.999,A -85,B 0,C 180,E1 -8304.736,E2 -8304.736} C_VEL
LIN {X 0,Y 453.464,Z 288.994,A -85,B 0,C 180,E1 -8307.942,E2 -8307.942} C_VEL
LIN {X 0,Y 453.457,Z 289.001,A -85,B 0,C 180,E1 -8310.761,E2 -8310.761} C_VEL
LIN {X 0,Y 453.469,Z 288.994,A -85,B 0,C 180,E1 -8313.913,E2 -8313.913} C_VEL
LIN {X 0,Y 453.452,Z 289.003,A -85,B 0,C 180,E1 -8317.19,E2 -8317.19} C_VEL
LIN {X 0,Y 453.473,Z 288.995,A -85,B 0,C 180,E1 -8320.611,E2 -8320.611} C_VEL
LIN {X 0,Y 453.484,Z 288.993,A -85,B 0,C 180,E1 -8324.528,E2 -8324.528} C_VEL
LIN {X 0,Y 453.438,Z 288.998,A -85,B 0,C 180,E1 -8328.071,E2 -8328.071} C_VEL
LIN {X 0,Y 453.445,Z 288.998,A -85,B 0,C 180,E1 -8330.801,E2 -8330.801} C_VEL
LIN {X 0,Y 453.45,Z 288.999,A -85,B 0,C 180,E1 -8333.916,E2 -8333.916} C_VEL
LIN {X 0,Y 453.477,Z 288.996,A -85,B 0,C 180,E1 -8337.15,E2 -8337.15} C_VEL
LIN {X 0,Y 453.469,Z 288.998,A -85,B 0,C 180,E1 -8340.267,E2 -8340.267} C_VEL
LIN {X 0,Y 453.529,Z 289.083,A -85,B 0,C 180,E1 -8343.295,E2 -8343.295} C_VEL
LIN {X 0,Y 455.927,Z 301.489,A -85,B 0,C 180,E1 -8345.609,E2 -8345.609} C_VEL
LIN {X 0,Y 455.3,Z 316.772,A -85,B 0,C 180,E1 -8348.255,E2 -8348.255} C_VEL
LIN {X 0,Y 454.491,Z 335.838,A -85,B 0,C 180,E1 -8351.518,E2 -8351.518} C_VEL
LIN {X 0,Y 454.2,Z 341.841,A -85,B 0,C 180,E1 -8352.537,E2 -8352.537} C_VEL
LIN {X 0,Y 457.351,Z 364.465,A -85,B 0,C 180,E1 -8353.024,E2 -8353.024} C_VEL
LIN {X 0,Y 456.602,Z 450.972,A -85,B 0,C 180,E1 -8354.402,E2 -8354.402} C_VEL
LIN {X 0,Y 456.207,Z 464.168,A -85,B 0,C 180,E1 -8354.789,E2 -8354.789} C_VEL
LIN {X 0,Y 455.734,Z 476.313,A -85,B 0,C 180,E1 -8355.315,E2 -8355.315} C_VEL
LIN {X 0,Y 455.187,Z 488.573,A -85,B 0,C 180,E1 -8356.039,E2 -8356.039} C_VEL
LIN {X 0,Y 454.637,Z 500.477,A -85,B 0,C 180,E1 -8356.957,E2 -8356.957} C_VEL
LIN {X 0,Y 454.09,Z 510.665,A -85,B 0,C 180,E1 -8357.939,E2 -8357.939} C_VEL
LIN {X 0,Y 453.616,Z 520.069,A -85,B 0,C 180,E1 -8359.059,E2 -8359.059} C_VEL
LIN {X 0,Y 453.163,Z 529.164,A -85,B 0,C 180,E1 -8360.402,E2 -8360.402} C_VEL
LIN {X 0,Y 452.851,Z 536.491,A -85,B 0,C 180,E1 -8361.746,E2 -8361.746} C_VEL
LIN {X 0,Y 452.674,Z 541.443,A -85,B 0,C 180,E1 -8362.865,E2 -8362.865} C_VEL
LIN {X 0,Y 452.557,Z 546.253,A -85,B 0,C 180,E1 -8364.206,E2 -8364.206} C_VEL
LIN {X 0,Y 452.488,Z 549.933,A -85,B 0,C 180,E1 -8365.545,E2 -8365.545} C_VEL
LIN {X 0,Y 452.489,Z 551.835,A -85,B 0,C 180,E1 -8366.438,E2 -8366.438} C_VEL
LIN {X 0,Y 452.522,Z 553.275,A -85,B 0,C 180,E1 -8367.329,E2 -8367.329} C_VEL
LIN {X 0,Y 452.489,Z 554.921,A -85,B 0,C 180,E1 -8369.109,E2 -8369.109} C_VEL
LIN {X 0,Y 452.468,Z 555.159,A -85,B 0,C 180,E1 -8369.999,E2 -8369.999} C_VEL
LIN {X 0,Y 452.489,Z 554.972,A -85,B 0,C 180,E1 -8370.889,E2 -8370.889} C_VEL
LIN {X 0,Y 452.523,Z 553.394,A -85,B 0,C 180,E1 -8372.67,E2 -8372.67} C_VEL
LIN {X 0,Y 452.491,Z 552.012,A -85,B 0,C 180,E1 -8373.561,E2 -8373.561} C_VEL
LIN {X 0,Y 452.545,Z 549.098,A -85,B 0,C 180,E1 -8374.899,E2 -8374.899} C_VEL
LIN {X 0,Y 452.61,Z 544.64,A -85,B 0,C 180,E1 -8376.395,E2 -8376.395} C_VEL
LIN {X 0,Y 452.776,Z 540.084,A -85,B 0,C 180,E1 -8377.581,E2 -8377.581} C_VEL
LIN {X 0,Y 452.997,Z 533.724,A -85,B 0,C 180,E1 -8378.925,E2 -8378.925} C_VEL
LIN {X 0,Y 453.39,Z 525.779,A -85,B 0,C 180,E1 -8380.268,E2 -8380.268} C_VEL
LIN {X 0,Y 453.989,Z 515.918,A -85,B 0,C 180,E1 -8381.609,E2 -8381.609} C_VEL
LIN {X 0,Y 454.487,Z 506.502,A -85,B 0,C 180,E1 -8382.646,E2 -8382.646} C_VEL
LIN {X 0,Y 455.081,Z 495.484,A -85,B 0,C 180,E1 -8383.621,E2 -8383.621} C_VEL
LIN {X 0,Y 455.661,Z 484.428,A -85,B 0,C 180,E1 -8384.4,E2 -8384.4} C_VEL
LIN {X 0,Y 456.268,Z 472.174,A -85,B 0,C 180,E1 -8385.065,E2 -8385.065} C_VEL
LIN {X 0,Y 456.788,Z 459.254,A -85,B 0,C 180,E1 -8385.562,E2 -8385.562} C_VEL
LIN {X 0,Y 457.144,Z 445.526,A -85,B 0,C 180,E1 -8385.893,E2 -8385.893} C_VEL
LIN {X 0,Y 457.817,Z 363.84,A -85,B 0,C 180,E1 -8387.193,E2 -8387.193} C_VEL
LIN {X 0,Y 454.428,Z 341.69,A -85,B 0,C 180,E1 -8387.703,E2 -8387.703} C_VEL
LIN {X 0,Y 455.214,Z 323.784,A -85,B 0,C 180,E1 -8390.799,E2 -8390.799} C_VEL
LIN {X 0,Y 456.149,Z 306.341,A -85,B 0,C 180,E1 -8393.855,E2 -8393.855} C_VEL
LIN {X 0,Y 456.134,Z 302.076,A -85,B 0,C 180,E1 -8394.624,E2 -8394.624} C_VEL
LIN {X 0,Y 454.04,Z 291.523,A -85,B 0,C 180,E1 -8396.672,E2 -8396.672} C_VEL
LIN {X 0,Y 453.495,Z 288.998,A -85,B 0,C 180,E1 -8397.204,E2 -8397.204} C_VEL
LIN {X 0,Y 453.467,Z 289.006,A -85,B 0,C 180,E1 -8399.783,E2 -8399.783} C_VEL
LIN {X 0,Y 453.482,Z 289,A -85,B 0,C 180,E1 -8403.187,E2 -8403.187} C_VEL
LIN {X 0,Y 453.448,Z 289.006,A -85,B 0,C 180,E1 -8406.298,E2 -8406.298} C_VEL
LIN {X 0,Y 453.464,Z 288.995,A -85,B 0,C 180,E1 -8409.452,E2 -8409.452} C_VEL
LIN {X 0,Y 453.474,Z 288.995,A -85,B 0,C 180,E1 -8411.934,E2 -8411.934} C_VEL
LIN {X 0,Y 453.482,Z 288.994,A -85,B 0,C 180,E1 -8415.471,E2 -8415.471} C_VEL
LIN {X 0,Y 453.476,Z 288.999,A -85,B 0,C 180,E1 -8418.209,E2 -8418.209} C_VEL
LIN {X 0,Y 453.512,Z 288.993,A -85,B 0,C 180,E1 -8420.79,E2 -8420.79} C_VEL
LIN {X 0,Y 453.451,Z 288.998,A -85,B 0,C 180,E1 -8423.917,E2 -8423.917} C_VEL
LIN {X 0,Y 453.475,Z 288.994,A -85,B 0,C 180,E1 -8427.151,E2 -8427.151} C_VEL
LIN {X 0,Y 453.471,Z 288.997,A -85,B 0,C 180,E1 -8430.268,E2 -8430.268} C_VEL
LIN {X 0,Y 453.498,Z 288.991,A -85,B 0,C 180,E1 -8433.293,E2 -8433.293} C_VEL
LIN {X 0,Y 453.494,Z 288.99,A -85,B 0,C 180,E1 -8436.238,E2 -8436.238} C_VEL
LIN {X 0,Y 453.479,Z 288.992,A -85,B 0,C 180,E1 -8439.118,E2 -8439.118} C_VEL
LIN {X 0,Y 453.508,Z 288.99,A -85,B 0,C 180,E1 -8441.945,E2 -8441.945} C_VEL
LIN {X 0,Y 453.537,Z 288.99,A -85,B 0,C 180,E1 -8444.726,E2 -8444.726} C_VEL
LIN {X 0,Y 453.556,Z 288.983,A -85,B 0,C 180,E1 -8448.379,E2 -8448.379} C_VEL
LIN {X 0,Y 453.648,Z 288.969,A -85,B 0,C 180,E1 -8451.985,E2 -8451.985} C_VEL
LIN {X 0,Y 453.667,Z 288.975,A -85,B 0,C 180,E1 -8454.667,E2 -8454.667} C_VEL
LIN {X 0,Y 453.762,Z 288.96,A -85,B 0,C 180,E1 -8457.337,E2 -8457.337} C_VEL
LIN {X 0,Y 453.821,Z 288.949,A -85,B 0,C 180,E1 -8460,E2 -8460} C_VEL
LIN {X 0,Y 453.762,Z 288.962,A -85,B 0,C 180,E1 -8462.663,E2 -8462.663} C_VEL
LIN {X 0,Y 453.674,Z 288.968,A -85,B 0,C 180,E1 -8466.226,E2 -8466.226} C_VEL
LIN {X 0,Y 453.589,Z 288.983,A -85,B 0,C 180,E1 -8468.914,E2 -8468.914} C_VEL
LIN {X 0,Y 453.56,Z 288.984,A -85,B 0,C 180,E1 -8472.529,E2 -8472.529} C_VEL
LIN {X 0,Y 453.541,Z 288.985,A -85,B 0,C 180,E1 -8476.196,E2 -8476.196} C_VEL
LIN {X 0,Y 453.515,Z 288.994,A -85,B 0,C 180,E1 -8479.04,E2 -8479.04} C_VEL
LIN {X 0,Y 453.474,Z 288.993,A -85,B 0,C 180,E1 -8481.837,E2 -8481.837} C_VEL
LIN {X 0,Y 453.498,Z 288.994,A -85,B 0,C 180,E1 -8484.736,E2 -8484.736} C_VEL
LIN {X 0,Y 453.529,Z 288.987,A -85,B 0,C 180,E1 -8487.96,E2 -8487.96} C_VEL
LIN {X 0,Y 453.463,Z 288.997,A -85,B 0,C 180,E1 -8491.526,E2 -8491.526} C_VEL
LIN {X 0,Y 453.481,Z 288.995,A -85,B 0,C 180,E1 -8494.777,E2 -8494.777} C_VEL
LIN {X 0,Y 453.457,Z 288.993,A -85,B 0,C 180,E1 -8498.313,E2 -8498.313} C_VEL
LIN {X 0,Y 453.492,Z 288.992,A -85,B 0,C 180,E1 -8500.61,E2 -8500.61} C_VEL
LIN {X 0,Y 453.458,Z 288.997,A -85,B 0,C 180,E1 -8504.223,E2 -8504.223} C_VEL
LIN {X 0,Y 453.436,Z 289.003,A -85,B 0,C 180,E1 -8507.003,E2 -8507.003} C_VEL
LIN {X 0,Y 453.47,Z 289.001,A -85,B 0,C 180,E1 -8509.413,E2 -8509.413} C_VEL
LIN {X 0,Y 453.44,Z 289.001,A -85,B 0,C 180,E1 -8512.81,E2 -8512.81} C_VEL
LIN {X 0,Y 453.469,Z 288.998,A -85,B 0,C 180,E1 -8516.087,E2 -8516.087} C_VEL
LIN {X 0,Y 453.468,Z 289.002,A -85,B 0,C 180,E1 -8519.241,E2 -8519.241} C_VEL
LIN {X 0,Y 453.525,Z 289.079,A -85,B 0,C 180,E1 -8520.592,E2 -8520.592} C_VEL
LIN {X 0,Y 454.786,Z 296.053,A -85,B 0,C 180,E1 -8522.086,E2 -8522.086} C_VEL
LIN {X 0,Y 454.727,Z 302.289,A -85,B 0,C 180,E1 -8523.341,E2 -8523.341} C_VEL
LIN {X 0,Y 458.201,Z 318.593,A -85,B 0,C 180,E1 -8523.777,E2 -8523.777} C_VEL
LIN {X 0,Y 457.222,Z 410.372,A -85,B 0,C 180,E1 -8525.257,E2 -8525.257} C_VEL
LIN {X 0,Y 456.954,Z 424.058,A -85,B 0,C 180,E1 -8525.676,E2 -8525.676} C_VEL
LIN {X 0,Y 456.511,Z 436.225,A -85,B 0,C 180,E1 -8526.225,E2 -8526.225} C_VEL
LIN {X 0,Y 456.019,Z 447.95,A -85,B 0,C 180,E1 -8526.943,E2 -8526.943} C_VEL
LIN {X 0,Y 455.098,Z 453.163,A -85,B 0,C 180,E1 -8527.3,E2 -8527.3} C_VEL
LIN {X 0,Y 451.889,Z 461.359,A -85,B 0,C 180,E1 -8527.888,E2 -8527.888} C_VEL
LIN {X 0,Y 448.69,Z 469.033,A -85,B 0,C 180,E1 -8528.559,E2 -8528.559} C_VEL
LIN {X 0,Y 447.775,Z 473.403,A -85,B 0,C 180,E1 -8529.036,E2 -8529.036} C_VEL
LIN {X 0,Y 447.183,Z 482.816,A -85,B 0,C 180,E1 -8530.3,E2 -8530.3} C_VEL
LIN {X 0,Y 446.62,Z 490.934,A -85,B 0,C 180,E1 -8531.657,E2 -8531.657} C_VEL
LIN {X 0,Y 446.222,Z 497.67,A -85,B 0,C 180,E1 -8533.06,E2 -8533.06} C_VEL
LIN {X 0,Y 445.887,Z 502.992,A -85,B 0,C 180,E1 -8534.458,E2 -8534.458} C_VEL
LIN {X 0,Y 445.677,Z 507.092,A -85,B 0,C 180,E1 -8535.853,E2 -8535.853} C_VEL
LIN {X 0,Y 445.555,Z 510.096,A -85,B 0,C 180,E1 -8537.243,E2 -8537.243} C_VEL
LIN {X 0,Y 445.501,Z 511.537,A -85,B 0,C 180,E1 -8538.166,E2 -8538.166} C_VEL
LIN {X 0,Y 445.422,Z 512.546,A -85,B 0,C 180,E1 -8539.086,E2 -8539.086} C_VEL
LIN {X 0,Y 445.363,Z 513.389,A -85,B 0,C 180,E1 -8540.921,E2 -8540.921} C_VEL
LIN {X 0,Y 445.38,Z 513.179,A -85,B 0,C 180,E1 -8541.836,E2 -8541.836} C_VEL
LIN {X 0,Y 445.513,Z 511.577,A -85,B 0,C 180,E1 -8543.661,E2 -8543.661} C_VEL
LIN {X 0,Y 445.536,Z 510.191,A -85,B 0,C 180,E1 -8544.57,E2 -8544.57} C_VEL
LIN {X 0,Y 445.627,Z 507.283,A -85,B 0,C 180,E1 -8545.931,E2 -8545.931} C_VEL
LIN {X 0,Y 445.806,Z 503.35,A -85,B 0,C 180,E1 -8547.29,E2 -8547.29} C_VEL
LIN {X 0,Y 445.971,Z 498.3,A -85,B 0,C 180,E1 -8548.646,E2 -8548.646} C_VEL
LIN {X 0,Y 446.409,Z 491.926,A -85,B 0,C 180,E1 -8550.001,E2 -8550.001} C_VEL
LIN {X 0,Y 446.795,Z 484.017,A -85,B 0,C 180,E1 -8551.353,E2 -8551.353} C_VEL
LIN {X 0,Y 447.236,Z 475.959,A -85,B 0,C 180,E1 -8552.477,E2 -8552.477} C_VEL
LIN {X 0,Y 447.706,Z 466.158,A -85,B 0,C 180,E1 -8553.601,E2 -8553.601} C_VEL
LIN {X 0,Y 448.291,Z 455.099,A -85,B 0,C 180,E1 -8554.609,E2 -8554.609} C_VEL
LIN {X 0,Y 448.882,Z 444.261,A -85,B 0,C 180,E1 -8555.391,E2 -8555.391} C_VEL
LIN {X 0,Y 449.197,Z 432.375,A -85,B 0,C 180,E1 -8556.063,E2 -8556.063} C_VEL
LIN {X 0,Y 449.555,Z 420.132,A -85,B 0,C 180,E1 -8556.565,E2 -8556.565} C_VEL
LIN {X 0,Y 449.875,Z 407.452,A -85,B 0,C 180,E1 -8556.898,E2 -8556.898} C_VEL
LIN {X 0,Y 450.734,Z 318.648,A -85,B 0,C 180,E1 -8558.321,E2 -8558.321} C_VEL
LIN {X 0,Y 447.623,Z 302.547,A -85,B 0,C 180,E1 -8558.699,E2 -8558.699} C_VEL
LIN {X 0,Y 447.405,Z 295.343,A -85,B 0,C 180,E1 -8560.179,E2 -8560.179} C_VEL
LIN {X 0,Y 446.512,Z 289.867,A -85,B 0,C 180,E1 -8561.376,E2 -8561.376} C_VEL
LIN {X 0,Y 446.466,Z 289.868,A -85,B 0,C 180,E1 -8563.658,E2 -8563.658} C_VEL
LIN {X 0,Y 446.493,Z 289.868,A -85,B 0,C 180,E1 -8566.46,E2 -8566.46} C_VEL
LIN {X 0,Y 446.474,Z 289.867,A -85,B 0,C 180,E1 -8569.304,E2 -8569.304} C_VEL
LIN {X 0,Y 446.422,Z 289.873,A -85,B 0,C 180,E1 -8572.2,E2 -8572.2} C_VEL
LIN {X 0,Y 446.434,Z 289.875,A -85,B 0,C 180,E1 -8575.154,E2 -8575.154} C_VEL
LIN {X 0,Y 446.422,Z 289.872,A -85,B 0,C 180,E1 -8578.184,E2 -8578.184} C_VEL
LIN {X 0,Y 446.412,Z 289.877,A -85,B 0,C 180,E1 -8581.301,E2 -8581.301} C_VEL
LIN {X 0,Y 446.427,Z 289.873,A -85,B 0,C 180,E1 -8584.524,E2 -8584.524} C_VEL
LIN {X 0,Y 446.415,Z 289.872,A -85,B 0,C 180,E1 -8588.078,E2 -8588.078} C_VEL
LIN {X 0,Y 446.405,Z 289.88,A -85,B 0,C 180,E1 -8591.394,E2 -8591.394} C_VEL
LIN {X 0,Y 446.454,Z 289.873,A -85,B 0,C 180,E1 -8595.104,E2 -8595.104} C_VEL
LIN {X 0,Y 446.405,Z 289.874,A -85,B 0,C 180,E1 -8598.606,E2 -8598.606} C_VEL
LIN {X 0,Y 446.407,Z 289.876,A -85,B 0,C 180,E1 -8601.923,E2 -8601.923} C_VEL
LIN {X 0,Y 446.427,Z 289.879,A -85,B 0,C 180,E1 -8605.476,E2 -8605.476} C_VEL
LIN {X 0,Y 446.419,Z 289.872,A -85,B 0,C 180,E1 -8608.699,E2 -8608.699} C_VEL
LIN {X 0,Y 446.454,Z 289.874,A -85,B 0,C 180,E1 -8611.83,E2 -8611.83} C_VEL
LIN {X 0,Y 446.424,Z 289.871,A -85,B 0,C 180,E1 -8614.845,E2 -8614.845} C_VEL
LIN {X 0,Y 446.454,Z 289.871,A -85,B 0,C 180,E1 -8618.245,E2 -8618.245} C_VEL
LIN {X 0,Y 446.453,Z 289.873,A -85,B 0,C 180,E1 -8621.649,E2 -8621.649} C_VEL
LIN {X 0,Y 446.511,Z 289.863,A -85,B 0,C 180,E1 -8624.48,E2 -8624.48} C_VEL
LIN {X 0,Y 446.511,Z 289.867,A -85,B 0,C 180,E1 -8628.193,E2 -8628.193} C_VEL
LIN {X 0,Y 446.515,Z 289.86,A -85,B 0,C 180,E1 -8630.944,E2 -8630.944} C_VEL
LIN {X 0,Y 446.61,Z 289.851,A -85,B 0,C 180,E1 -8633.676,E2 -8633.676} C_VEL
LIN {X 0,Y 446.657,Z 289.842,A -85,B 0,C 180,E1 -8637.294,E2 -8637.294} C_VEL
LIN {X 0,Y 446.721,Z 289.839,A -85,B 0,C 180,E1 -8640,E2 -8640} C_VEL
LIN {X 0,Y 446.655,Z 289.846,A -85,B 0,C 180,E1 -8642.705,E2 -8642.705} C_VEL
LIN {X 0,Y 446.609,Z 289.855,A -85,B 0,C 180,E1 -8646.324,E2 -8646.324} C_VEL
LIN {X 0,Y 446.509,Z 289.862,A -85,B 0,C 180,E1 -8649.056,E2 -8649.056} C_VEL
LIN {X 0,Y 446.526,Z 289.865,A -85,B 0,C 180,E1 -8652.729,E2 -8652.729} C_VEL
LIN {X 0,Y 446.488,Z 289.869,A -85,B 0,C 180,E1 -8656.459,E2 -8656.459} C_VEL
LIN {X 0,Y 446.472,Z 289.867,A -85,B 0,C 180,E1 -8659.303,E2 -8659.303} C_VEL
LIN {X 0,Y 446.42,Z 289.873,A -85,B 0,C 180,E1 -8662.199,E2 -8662.199} C_VEL
LIN {X 0,Y 446.432,Z 289.875,A -85,B 0,C 180,E1 -8665.154,E2 -8665.154} C_VEL
LIN {X 0,Y 446.419,Z 289.873,A -85,B 0,C 180,E1 -8668.183,E2 -8668.183} C_VEL
LIN {X 0,Y 446.41,Z 289.877,A -85,B 0,C 180,E1 -8671.301,E2 -8671.301} C_VEL
LIN {X 0,Y 446.425,Z 289.873,A -85,B 0,C 180,E1 -8674.523,E2 -8674.523} C_VEL
LIN {X 0,Y 446.413,Z 289.873,A -85,B 0,C 180,E1 -8678.078,E2 -8678.078} C_VEL
LIN {X 0,Y 446.402,Z 289.88,A -85,B 0,C 180,E1 -8681.394,E2 -8681.394} C_VEL
LIN {X 0,Y 446.452,Z 289.874,A -85,B 0,C 180,E1 -8685.104,E2 -8685.104} C_VEL
LIN {X 0,Y 446.402,Z 289.875,A -85,B 0,C 180,E1 -8688.605,E2 -8688.605} C_VEL
LIN {X 0,Y 446.404,Z 289.876,A -85,B 0,C 180,E1 -8691.923,E2 -8691.923} C_VEL
LIN {X 0,Y 446.425,Z 289.88,A -85,B 0,C 180,E1 -8695.476,E2 -8695.476} C_VEL
LIN {X 0,Y 446.417,Z 289.872,A -85,B 0,C 180,E1 -8698.699,E2 -8698.699} C_VEL
LIN {X 0,Y 446.451,Z 289.874,A -85,B 0,C 180,E1 -8701.83,E2 -8701.83} C_VEL
LIN {X 0,Y 446.487,Z 289.923,A -85,B 0,C 180,E1 -8703.098,E2 -8703.098} C_VEL
LIN {X 0,Y 448.978,Z 303.391,A -85,B 0,C 180,E1 -8705.645,E2 -8705.645} C_VEL
LIN {X 0,Y 448.245,Z 318.971,A -85,B 0,C 180,E1 -8708.379,E2 -8708.379} C_VEL
LIN {X 0,Y 447.463,Z 336.684,A -85,B 0,C 180,E1 -8711.454,E2 -8711.454} C_VEL
LIN {X 0,Y 447.22,Z 341.767,A -85,B 0,C 180,E1 -8712.308,E2 -8712.308} C_VEL
LIN {X 0,Y 450.483,Z 364.14,A -85,B 0,C 180,E1 -8712.787,E2 -8712.787} C_VEL
LIN {X 0,Y 449.733,Z 450.67,A -85,B 0,C 180,E1 -8714.187,E2 -8714.187} C_VEL
LIN {X 0,Y 449.311,Z 463.86,A -85,B 0,C 180,E1 -8714.578,E2 -8714.578} C_VEL
LIN {X 0,Y 448.801,Z 476.573,A -85,B 0,C 180,E1 -8715.141,E2 -8715.141} C_VEL
LIN {X 0,Y 448.242,Z 487.863,A -85,B 0,C 180,E1 -8715.818,E2 -8715.818} C_VEL
LIN {X 0,Y 447.668,Z 499.749,A -85,B 0,C 180,E1 -8716.742,E2 -8716.742} C_VEL
LIN {X 0,Y 447.101,Z 510.086,A -85,B 0,C 180,E1 -8717.748,E2 -8717.748} C_VEL
LIN {X 0,Y 446.618,Z 519.555,A -85,B 0,C 180,E1 -8718.885,E2 -8718.885} C_VEL
LIN {X 0,Y 446.122,Z 528.683,A -85,B 0,C 180,E1 -8720.249,E2 -8720.249} C_VEL
LIN {X 0,Y 445.792,Z 536.039,A -85,B 0,C 180,E1 -8721.614,E2 -8721.614} C_VEL
LIN {X 0,Y 445.603,Z 541.016,A -85,B 0,C 180,E1 -8722.751,E2 -8722.751} C_VEL
LIN {X 0,Y 445.483,Z 545.295,A -85,B 0,C 180,E1 -8723.939,E2 -8723.939} C_VEL
LIN {X 0,Y 445.414,Z 549.548,A -85,B 0,C 180,E1 -8725.475,E2 -8725.475} C_VEL
LIN {X 0,Y 445.39,Z 551.459,A -85,B 0,C 180,E1 -8726.381,E2 -8726.381} C_VEL
LIN {X 0,Y 445.446,Z 552.917,A -85,B 0,C 180,E1 -8727.286,E2 -8727.286} C_VEL
LIN {X 0,Y 445.396,Z 554.578,A -85,B 0,C 180,E1 -8729.095,E2 -8729.095} C_VEL
LIN {X 0,Y 445.404,Z 554.826,A -85,B 0,C 180,E1 -8729.999,E2 -8729.999} C_VEL
LIN {X 0,Y 445.396,Z 554.653,A -85,B 0,C 180,E1 -8730.904,E2 -8730.904} C_VEL
LIN {X 0,Y 445.447,Z 553.091,A -85,B 0,C 180,E1 -8732.712,E2 -8732.712} C_VEL
LIN {X 0,Y 445.391,Z 551.717,A -85,B 0,C 180,E1 -8733.618,E2 -8733.618} C_VEL
LIN {X 0,Y 445.473,Z 548.822,A -85,B 0,C 180,E1 -8734.977,E2 -8734.977} C_VEL
LIN {X 0,Y 445.529,Z 544.752,A -85,B 0,C 180,E1 -8736.385,E2 -8736.385} C_VEL
LIN {X 0,Y 445.708,Z 539.848,A -85,B 0,C 180,E1 -8737.702,E2 -8737.702} C_VEL
LIN {X 0,Y 445.955,Z 533.52,A -85,B 0,C 180,E1 -8739.067,E2 -8739.067} C_VEL
LIN {X 0,Y 446.353,Z 525.615,A -85,B 0,C 180,E1 -8740.432,E2 -8740.432} C_VEL
LIN {X 0,Y 446.919,Z 517.579,A -85,B 0,C 180,E1 -8741.566,E2 -8741.566} C_VEL
LIN {X 0,Y 447.453,Z 507.792,A -85,B 0,C 180,E1 -8742.702,E2 -8742.702} C_VEL
LIN {X 0,Y 448.116,Z 496.915,A -85,B 0,C 180,E1 -8743.721,E2 -8743.721} C_VEL
LIN {X 0,Y 448.796,Z 484.53,A -85,B 0,C 180,E1 -8744.626,E2 -8744.626} C_VEL
LIN {X 0,Y 449.444,Z 472.407,A -85,B 0,C 180,E1 -8745.3,E2 -8745.3} C_VEL
LIN {X 0,Y 449.989,Z 459.841,A -85,B 0,C 180,E1 -8745.803,E2 -8745.803} C_VEL
LIN {X 0,Y 450.36,Z 446.715,A -85,B 0,C 180,E1 -8746.138,E2 -8746.138} C_VEL
LIN {X 0,Y 451.026,Z 363.732,A -85,B 0,C 180,E1 -8747.488,E2 -8747.488} C_VEL
LIN {X 0,Y 447.487,Z 341.229,A -85,B 0,C 180,E1 -8748.04,E2 -8748.04} C_VEL
LIN {X 0,Y 448.571,Z 320.96,A -85,B 0,C 180,E1 -8751.603,E2 -8751.603} C_VEL
LIN {X 0,Y 449.38,Z 305.166,A -85,B 0,C 180,E1 -8754.429,E2 -8754.429} C_VEL
LIN {X 0,Y 447.946,Z 296.789,A -85,B 0,C 180,E1 -8756.059,E2 -8756.059} C_VEL
LIN {X 0,Y 446.466,Z 289.875,A -85,B 0,C 180,E1 -8757.478,E2 -8757.478} C_VEL
LIN {X 0,Y 446.424,Z 289.885,A -85,B 0,C 180,E1 -8760.249,E2 -8760.249} C_VEL
LIN {X 0,Y 446.444,Z 289.877,A -85,B 0,C 180,E1 -8763.453,E2 -8763.453} C_VEL
LIN {X 0,Y 446.398,Z 289.88,A -85,B 0,C 180,E1 -8766.745,E2 -8766.745} C_VEL
LIN {X 0,Y 446.434,Z 289.876,A -85,B 0,C 180,E1 -8770.198,E2 -8770.198} C_VEL
LIN {X 0,Y 446.426,Z 289.878,A -85,B 0,C 180,E1 -8772.604,E2 -8772.604} C_VEL
LIN {X 0,Y 446.449,Z 289.871,A -85,B 0,C 180,E1 -8775.103,E2 -8775.103} C_VEL
LIN {X 0,Y 446.425,Z 289.876,A -85,B 0,C 180,E1 -8778.609,E2 -8778.609} C_VEL
LIN {X 0,Y 446.456,Z 289.87,A -85,B 0,C 180,E1 -8780.974,E2 -8780.974} C_VEL
LIN {X 0,Y 446.414,Z 289.879,A -85,B 0,C 180,E1 -8784.374,E2 -8784.374} C_VEL
LIN {X 0,Y 446.416,Z 289.872,A -85,B 0,C 180,E1 -8787.638,E2 -8787.638} C_VEL
LIN {X 0,Y 446.445,Z 289.873,A -85,B 0,C 180,E1 -8790.79,E2 -8790.79} C_VEL
LIN {X 0,Y 446.474,Z 289.865,A -85,B 0,C 180,E1 -8793.848,E2 -8793.848} C_VEL
LIN {X 0,Y 446.423,Z 289.878,A -85,B 0,C 180,E1 -8796.823,E2 -8796.823} C_VEL
LIN {X 0,Y 446.441,Z 289.865,A -85,B 0,C 180,E1 -8799.737,E2 -8799.737} C_VEL
LIN {X 0,Y 446.461,Z 289.874,A -85,B 0,C 180,E1 -8802.597,E2 -8802.597} C_VEL
LIN {X 0,Y 446.469,Z 289.868,A -85,B 0,C 180,E1 -8805.412,E2 -8805.412} C_VEL
LIN {X 0,Y 446.514,Z 289.858,A -85,B 0,C 180,E1 -8808.193,E2 -8808.193} C_VEL
LIN {X 0,Y 446.597,Z 289.847,A -85,B 0,C 180,E1 -8811.858,E2 -8811.858} C_VEL
LIN {X 0,Y 446.642,Z 289.849,A -85,B 0,C 180,E1 -8814.583,E2 -8814.583} C_VEL
LIN {X 0,Y 446.706,Z 289.84,A -85,B 0,C 180,E1 -8817.295,E2 -8817.295} C_VEL
LIN {X 0,Y 446.791,Z 289.824,A -85,B 0,C 180,E1 -8820,E2 -8820} C_VEL
LIN {X 0,Y 446.705,Z 289.841,A -85,B 0,C 180,E1 -8822.706,E2 -8822.706} C_VEL
LIN {X 0,Y 446.644,Z 289.844,A -85,B 0,C 180,E1 -8826.324,E2 -8826.324} C_VEL
LIN {X 0,Y 446.535,Z 289.861,A -85,B 0,C 180,E1 -8829.056,E2 -8829.056} C_VEL
LIN {X 0,Y 446.518,Z 289.864,A -85,B 0,C 180,E1 -8832.73,E2 -8832.73} C_VEL
LIN {X 0,Y 446.493,Z 289.863,A -85,B 0,C 180,E1 -8836.228,E2 -8836.228} C_VEL
LIN {X 0,Y 446.466,Z 289.873,A -85,B 0,C 180,E1 -8839.304,E2 -8839.304} C_VEL
LIN {X 0,Y 446.415,Z 289.872,A -85,B 0,C 180,E1 -8842.2,E2 -8842.2} C_VEL
LIN {X 0,Y 446.441,Z 289.874,A -85,B 0,C 180,E1 -8845.154,E2 -8845.154} C_VEL
LIN {X 0,Y 446.483,Z 289.864,A -85,B 0,C 180,E1 -8848.179,E2 -8848.179} C_VEL
LIN {X 0,Y 446.416,Z 289.872,A -85,B 0,C 180,E1 -8851.775,E2 -8851.775} C_VEL
LIN {X 0,Y 446.421,Z 289.873,A -85,B 0,C 180,E1 -8854.524,E2 -8854.524} C_VEL
LIN {X 0,Y 446.411,Z 289.871,A -85,B 0,C 180,E1 -8858.079,E2 -8858.079} C_VEL
LIN {X 0,Y 446.414,Z 289.878,A -85,B 0,C 180,E1 -8861.393,E2 -8861.393} C_VEL
LIN {X 0,Y 446.449,Z 289.875,A -85,B 0,C 180,E1 -8865.105,E2 -8865.105} C_VEL
LIN {X 0,Y 446.405,Z 289.877,A -85,B 0,C 180,E1 -8868.607,E2 -8868.607} C_VEL
LIN {X 0,Y 446.402,Z 289.879,A -85,B 0,C 180,E1 -8871.924,E2 -8871.924} C_VEL
LIN {X 0,Y 446.423,Z 289.876,A -85,B 0,C 180,E1 -8875.477,E2 -8875.477} C_VEL
LIN {X 0,Y 446.413,Z 289.878,A -85,B 0,C 180,E1 -8878.7,E2 -8878.7} C_VEL
LIN {X 0,Y 446.473,Z 290.013,A -85,B 0,C 180,E1 -8880.353,E2 -8880.353} C_VEL
LIN {X 0,Y 447.863,Z 297.176,A -85,B 0,C 180,E1 -8881.916,E2 -8881.916} C_VEL
LIN {X 0,Y 447.831,Z 302.633,A -85,B 0,C 180,E1 -8883.03,E2 -8883.03} C_VEL
LIN {X 0,Y 451.526,Z 319.586,A -85,B 0,C 180,E1 -8883.493,E2 -8883.493} C_VEL
LIN {X 0,Y 450.48,Z 410.882,A -85,B 0,C 180,E1 -8884.988,E2 -8884.988} C_VEL
LIN {X 0,Y 450.191,Z 424.403,A -85,B 0,C 180,E1 -8885.41,E2 -8885.41} C_VEL
LIN {X 0,Y 449.722,Z 436.561,A -85,B 0,C 180,E1 -8885.966,E2 -8885.966} C_VEL
LIN {X 0,Y 449.168,Z 448.768,A -85,B 0,C 180,E1 -8886.73,E2 -8886.73} C_VEL
LIN {X 0,Y 448.613,Z 459.21,A -85,B 0,C 180,E1 -8887.564,E2 -8887.564} C_VEL
LIN {X 0,Y 447.968,Z 469.727,A -85,B 0,C 180,E1 -8888.608,E2 -8888.608} C_VEL
LIN {X 0,Y 447.775,Z 473.403,A -85,B 0,C 180,E1 -8889.036,E2 -8889.036} C_VEL
LIN {X 0,Y 446.855,Z 477.694,A -85,B 0,C 180,E1 -8889.544,E2 -8889.544} C_VEL
LIN {X 0,Y 443.612,Z 484.362,A -85,B 0,C 180,E1 -8890.394,E2 -8890.394} C_VEL
LIN {X 0,Y 440.384,Z 490.396,A -85,B 0,C 180,E1 -8891.324,E2 -8891.324} C_VEL
LIN {X 0,Y 439.498,Z 493.691,A -85,B 0,C 180,E1 -8891.952,E2 -8891.952} C_VEL
LIN {X 0,Y 439.116,Z 499.449,A -85,B 0,C 180,E1 -8893.257,E2 -8893.257} C_VEL
LIN {X 0,Y 438.796,Z 504.436,A -85,B 0,C 180,E1 -8894.677,E2 -8894.677} C_VEL
LIN {X 0,Y 438.576,Z 508.25,A -85,B 0,C 180,E1 -8896.092,E2 -8896.092} C_VEL
LIN {X 0,Y 438.483,Z 510.202,A -85,B 0,C 180,E1 -8897.033,E2 -8897.033} C_VEL
LIN {X 0,Y 438.425,Z 511.722,A -85,B 0,C 180,E1 -8897.973,E2 -8897.973} C_VEL
LIN {X 0,Y 438.341,Z 512.777,A -85,B 0,C 180,E1 -8898.908,E2 -8898.908} C_VEL
LIN {X 0,Y 438.276,Z 513.702,A -85,B 0,C 180,E1 -8900.773,E2 -8900.773} C_VEL
LIN {X 0,Y 438.292,Z 513.57,A -85,B 0,C 180,E1 -8901.703,E2 -8901.703} C_VEL
LIN {X 0,Y 438.425,Z 512.049,A -85,B 0,C 180,E1 -8903.558,E2 -8903.558} C_VEL
LIN {X 0,Y 438.448,Z 510.71,A -85,B 0,C 180,E1 -8904.482,E2 -8904.482} C_VEL
LIN {X 0,Y 438.516,Z 507.882,A -85,B 0,C 180,E1 -8905.865,E2 -8905.865} C_VEL
LIN {X 0,Y 438.744,Z 504.033,A -85,B 0,C 180,E1 -8907.246,E2 -8907.246} C_VEL
LIN {X 0,Y 438.9,Z 499.084,A -85,B 0,C 180,E1 -8908.624,E2 -8908.624} C_VEL
LIN {X 0,Y 439.355,Z 492.85,A -85,B 0,C 180,E1 -8910.001,E2 -8910.001} C_VEL
LIN {X 0,Y 439.753,Z 485.077,A -85,B 0,C 180,E1 -8911.374,E2 -8911.374} C_VEL
LIN {X 0,Y 440.295,Z 475.404,A -85,B 0,C 180,E1 -8912.745,E2 -8912.745} C_VEL
LIN {X 0,Y 440.819,Z 465.362,A -85,B 0,C 180,E1 -8913.886,E2 -8913.886} C_VEL
LIN {X 0,Y 441.421,Z 454.004,A -85,B 0,C 180,E1 -8914.91,E2 -8914.91} C_VEL
LIN {X 0,Y 442.081,Z 442.815,A -85,B 0,C 180,E1 -8915.703,E2 -8915.703} C_VEL
LIN {X 0,Y 442.363,Z 431.536,A -85,B 0,C 180,E1 -8916.328,E2 -8916.328} C_VEL
LIN {X 0,Y 442.736,Z 418.6,A -85,B 0,C 180,E1 -8916.838,E2 -8916.838} C_VEL
LIN {X 0,Y 443.036,Z 406.2,A -85,B 0,C 180,E1 -8917.148,E2 -8917.148} C_VEL
LIN {X 0,Y 443.887,Z 319.456,A -85,B 0,C 180,E1 -8918.555,E2 -8918.555} C_VEL
LIN {X 0,Y 440.635,Z 302.716,A -85,B 0,C 180,E1 -8918.98,E2 -8918.98} C_VEL
LIN {X 0,Y 440.537,Z 297.27,A -85,B 0,C 180,E1 -8920.108,E2 -8920.108} C_VEL
LIN {X 0,Y 439.489,Z 290.742,A -85,B 0,C 180,E1 -8921.531,E2 -8921.531} C_VEL
LIN {X 0,Y 439.449,Z 290.746,A -85,B 0,C 180,E1 -8924.827,E2 -8924.827} C_VEL
LIN {X 0,Y 439.406,Z 290.746,A -85,B 0,C 180,E1 -8927.692,E2 -8927.692} C_VEL
LIN {X 0,Y 439.393,Z 290.753,A -85,B 0,C 180,E1 -8930.603,E2 -8930.603} C_VEL
LIN {X 0,Y 439.371,Z 290.751,A -85,B 0,C 180,E1 -8933.572,E2 -8933.572} C_VEL
LIN {X 0,Y 439.37,Z 290.754,A -85,B 0,C 180,E1 -8936.608,E2 -8936.608} C_VEL
LIN {X 0,Y 439.374,Z 290.75,A -85,B 0,C 180,E1 -8939.727,E2 -8939.727} C_VEL
LIN {X 0,Y 439.376,Z 290.757,A -85,B 0,C 180,E1 -8942.946,E2 -8942.946} C_VEL
LIN {X 0,Y 439.377,Z 290.75,A -85,B 0,C 180,E1 -8946.288,E2 -8946.288} C_VEL
LIN {X 0,Y 439.364,Z 290.752,A -85,B 0,C 180,E1 -8949.78,E2 -8949.78} C_VEL
LIN {X 0,Y 439.338,Z 290.755,A -85,B 0,C 180,E1 -8952.62,E2 -8952.62} C_VEL
LIN {X 0,Y 439.402,Z 290.754,A -85,B 0,C 180,E1 -8955.27,E2 -8955.27} C_VEL
LIN {X 0,Y 439.358,Z 290.755,A -85,B 0,C 180,E1 -8959.016,E2 -8959.016} C_VEL
LIN {X 0,Y 439.343,Z 290.754,A -85,B 0,C 180,E1 -8962.564,E2 -8962.564} C_VEL
LIN {X 0,Y 439.399,Z 290.747,A -85,B 0,C 180,E1 -8964.843,E2 -8964.843} C_VEL
LIN {X 0,Y 439.374,Z 290.751,A -85,B 0,C 180,E1 -8968.139,E2 -8968.139} C_VEL
LIN {X 0,Y 439.409,Z 290.753,A -85,B 0,C 180,E1 -8971.605,E2 -8971.605} C_VEL
LIN {X 0,Y 439.37,Z 290.751,A -85,B 0,C 180,E1 -8974.412,E2 -8974.412} C_VEL
LIN {X 0,Y 439.369,Z 290.754,A -85,B 0,C 180,E1 -8977.424,E2 -8977.424} C_VEL
LIN {X 0,Y 439.446,Z 290.741,A -85,B 0,C 180,E1 -8980.663,E2 -8980.663} C_VEL
LIN {X 0,Y 439.466,Z 290.743,A -85,B 0,C 180,E1 -8984.224,E2 -8984.224} C_VEL
LIN {X 0,Y 439.48,Z 290.745,A -85,B 0,C 180,E1 -8988.001,E2 -8988.001} C_VEL
LIN {X 0,Y 439.485,Z 290.739,A -85,B 0,C 180,E1 -8991.725,E2 -8991.725} C_VEL
LIN {X 0,Y 439.601,Z 290.725,A -85,B 0,C 180,E1 -8994.495,E2 -8994.495} C_VEL
LIN {X 0,Y 439.631,Z 290.725,A -85,B 0,C 180,E1 -8998.168,E2 -8998.168} C_VEL
LIN {X 0,Y 439.673,Z 290.717,A -85,B 0,C 180,E1 -9000,E2 -9000} C_VEL
LIN {X 0,Y 439.606,Z 290.724,A -85,B 0,C 180,E1 -9002.749,E2 -9002.749} C_VEL
LIN {X 0,Y 439.562,Z 290.735,A -85,B 0,C 180,E1 -9006.426,E2 -9006.426} C_VEL
LIN {X 0,Y 439.476,Z 290.738,A -85,B 0,C 180,E1 -9009.202,E2 -9009.202} C_VEL
LIN {X 0,Y 439.469,Z 290.741,A -85,B 0,C 180,E1 -9012.937,E2 -9012.937} C_VEL
LIN {X 0,Y 439.448,Z 290.745,A -85,B 0,C 180,E1 -9016.347,E2 -9016.347} C_VEL
LIN {X 0,Y 439.405,Z 290.746,A -85,B 0,C 180,E1 -9019.626,E2 -9019.626} C_VEL
LIN {X 0,Y 439.365,Z 290.756,A -85,B 0,C 180,E1 -9022.575,E2 -9022.575} C_VEL
LIN {X 0,Y 439.373,Z 290.75,A -85,B 0,C 180,E1 -9025.587,E2 -9025.587} C_VEL
LIN {X 0,Y 439.384,Z 290.753,A -85,B 0,C 180,E1 -9028.676,E2 -9028.676} C_VEL
LIN {X 0,Y 439.365,Z 290.751,A -85,B 0,C 180,E1 -9032.028,E2 -9032.028} C_VEL
LIN {X 0,Y 439.394,Z 290.752,A -85,B 0,C 180,E1 -9035.339,E2 -9035.339} C_VEL
LIN {X 0,Y 439.365,Z 290.753,A -85,B 0,C 180,E1 -9038.597,E2 -9038.597} C_VEL
LIN {X 0,Y 439.351,Z 290.753,A -85,B 0,C 180,E1 -9042.21,E2 -9042.21} C_VEL
LIN {X 0,Y 439.4,Z 290.755,A -85,B 0,C 180,E1 -9045.27,E2 -9045.27} C_VEL
LIN {X 0,Y 439.355,Z 290.756,A -85,B 0,C 180,E1 -9049.016,E2 -9049.016} C_VEL
LIN {X 0,Y 439.341,Z 290.754,A -85,B 0,C 180,E1 -9052.563,E2 -9052.563} C_VEL
LIN {X 0,Y 439.397,Z 290.748,A -85,B 0,C 180,E1 -9054.843,E2 -9054.843} C_VEL
LIN {X 0,Y 439.372,Z 290.754,A -85,B 0,C 180,E1 -9058.139,E2 -9058.139} C_VEL
LIN {X 0,Y 439.406,Z 290.753,A -85,B 0,C 180,E1 -9061.605,E2 -9061.605} C_VEL
LIN {X 0,Y 439.435,Z 290.866,A -85,B 0,C 180,E1 -9062.915,E2 -9062.915} C_VEL
LIN {X 0,Y 441.777,Z 302.931,A -85,B 0,C 180,E1 -9065.244,E2 -9065.244} C_VEL
LIN {X 0,Y 441.943,Z 306.103,A -85,B 0,C 180,E1 -9065.827,E2 -9065.827} C_VEL
LIN {X 0,Y 441.134,Z 322.532,A -85,B 0,C 180,E1 -9068.749,E2 -9068.749} C_VEL
LIN {X 0,Y 440.356,Z 339.004,A -85,B 0,C 180,E1 -9071.65,E2 -9071.65} C_VEL
LIN {X 0,Y 440.252,Z 341.456,A -85,B 0,C 180,E1 -9072.054,E2 -9072.054} C_VEL
LIN {X 0,Y 443.64,Z 365.408,A -85,B 0,C 180,E1 -9072.571,E2 -9072.571} C_VEL
LIN {X 0,Y 442.86,Z 450.273,A -85,B 0,C 180,E1 -9073.964,E2 -9073.964} C_VEL
LIN {X 0,Y 442.43,Z 463.491,A -85,B 0,C 180,E1 -9074.362,E2 -9074.362} C_VEL
LIN {X 0,Y 441.915,Z 475.65,A -85,B 0,C 180,E1 -9074.904,E2 -9074.904} C_VEL
LIN {X 0,Y 441.324,Z 487.111,A -85,B 0,C 180,E1 -9075.591,E2 -9075.591} C_VEL
LIN {X 0,Y 440.711,Z 499.135,A -85,B 0,C 180,E1 -9076.534,E2 -9076.534} C_VEL
LIN {X 0,Y 440.126,Z 509.484,A -85,B 0,C 180,E1 -9077.55,E2 -9077.55} C_VEL
LIN {X 0,Y 439.609,Z 519.017,A -85,B 0,C 180,E1 -9078.706,E2 -9078.706} C_VEL
LIN {X 0,Y 439.055,Z 528.183,A -85,B 0,C 180,E1 -9080.091,E2 -9080.091} C_VEL
LIN {X 0,Y 438.722,Z 535.572,A -85,B 0,C 180,E1 -9081.478,E2 -9081.478} C_VEL
LIN {X 0,Y 438.529,Z 540.577,A -85,B 0,C 180,E1 -9082.633,E2 -9082.633} C_VEL
LIN {X 0,Y 438.383,Z 545.311,A -85,B 0,C 180,E1 -9083.979,E2 -9083.979} C_VEL
LIN {X 0,Y 438.344,Z 549.157,A -85,B 0,C 180,E1 -9085.401,E2 -9085.401} C_VEL
LIN {X 0,Y 438.293,Z 551.077,A -85,B 0,C 180,E1 -9086.322,E2 -9086.322} C_VEL
LIN {X 0,Y 438.371,Z 552.556,A -85,B 0,C 180,E1 -9087.243,E2 -9087.243} C_VEL
LIN {X 0,Y 438.306,Z 554.234,A -85,B 0,C 180,E1 -9089.081,E2 -9089.081} C_VEL
LIN {X 0,Y 438.312,Z 554.491,A -85,B 0,C 180,E1 -9089.999,E2 -9089.999} C_VEL
LIN {X 0,Y 438.306,Z 554.336,A -85,B 0,C 180,E1 -9090.918,E2 -9090.918} C_VEL
LIN {X 0,Y 438.372,Z 552.793,A -85,B 0,C 180,E1 -9092.756,E2 -9092.756} C_VEL
LIN {X 0,Y 438.292,Z 551.426,A -85,B 0,C 180,E1 -9093.677,E2 -9093.677} C_VEL
LIN {X 0,Y 438.382,Z 548.552,A -85,B 0,C 180,E1 -9095.058,E2 -9095.058} C_VEL
LIN {X 0,Y 438.447,Z 544.649,A -85,B 0,C 180,E1 -9096.442,E2 -9096.442} C_VEL
LIN {X 0,Y 438.639,Z 539.624,A -85,B 0,C 180,E1 -9097.827,E2 -9097.827} C_VEL
LIN {X 0,Y 438.926,Z 533.328,A -85,B 0,C 180,E1 -9099.213,E2 -9099.213} C_VEL
LIN {X 0,Y 439.34,Z 525.467,A -85,B 0,C 180,E1 -9100.6,E2 -9100.6} C_VEL
LIN {X 0,Y 440.041,Z 515.687,A -85,B 0,C 180,E1 -9101.983,E2 -9101.983} C_VEL
LIN {X 0,Y 440.587,Z 506.15,A -85,B 0,C 180,E1 -9103.077,E2 -9103.077} C_VEL
LIN {X 0,Y 441.275,Z 495.542,A -85,B 0,C 180,E1 -9104.056,E2 -9104.056} C_VEL
LIN {X 0,Y 442.008,Z 482.906,A -85,B 0,C 180,E1 -9104.973,E2 -9104.973} C_VEL
LIN {X 0,Y 442.733,Z 470.318,A -85,B 0,C 180,E1 -9105.655,E2 -9105.655} C_VEL
LIN {X 0,Y 443.312,Z 456.862,A -85,B 0,C 180,E1 -9106.166,E2 -9106.166} C_VEL
LIN {X 0,Y 443.686,Z 443.484,A -85,B 0,C 180,E1 -9106.477,E2 -9106.477} C_VEL
LIN {X 0,Y 444.351,Z 364.783,A -85,B 0,C 180,E1 -9107.769,E2 -9107.769} C_VEL
LIN {X 0,Y 440.549,Z 340.991,A -85,B 0,C 180,E1 -9108.351,E2 -9108.351} C_VEL
LIN {X 0,Y 441.625,Z 322.168,A -85,B 0,C 180,E1 -9111.715,E2 -9111.715} C_VEL
LIN {X 0,Y 442.426,Z 307.429,A -85,B 0,C 180,E1 -9114.394,E2 -9114.394} C_VEL
LIN {X 0,Y 441.817,Z 302.054,A -85,B 0,C 180,E1 -9115.435,E2 -9115.435} C_VEL
LIN {X 0,Y 439.452,Z 290.75,A -85,B 0,C 180,E1 -9117.748,E2 -9117.748} C_VEL
LIN {X 0,Y 439.359,Z 290.763,A -85,B 0,C 180,E1 -9120.788,E2 -9120.788} C_VEL
LIN {X 0,Y 439.383,Z 290.759,A -85,B 0,C 180,E1 -9124.043,E2 -9124.043} C_VEL
LIN {X 0,Y 439.344,Z 290.758,A -85,B 0,C 180,E1 -9126.886,E2 -9126.886} C_VEL
LIN {X 0,Y 439.399,Z 290.749,A -85,B 0,C 180,E1 -9129.849,E2 -9129.849} C_VEL
LIN {X 0,Y 439.379,Z 290.756,A -85,B 0,C 180,E1 -9132.626,E2 -9132.626} C_VEL
LIN {X 0,Y 439.397,Z 290.749,A -85,B 0,C 180,E1 -9135.27,E2 -9135.27} C_VEL
LIN {X 0,Y 439.385,Z 290.752,A -85,B 0,C 180,E1 -9138.743,E2 -9138.743} C_VEL
LIN {X 0,Y 439.374,Z 290.749,A -85,B 0,C 180,E1 -9141.607,E2 -9141.607} C_VEL
LIN {X 0,Y 439.393,Z 290.749,A -85,B 0,C 180,E1 -9144.843,E2 -9144.843} C_VEL
LIN {X 0,Y 439.369,Z 290.752,A -85,B 0,C 180,E1 -9148.139,E2 -9148.139} C_VEL
LIN {X 0,Y 439.429,Z 290.74,A -85,B 0,C 180,E1 -9151.598,E2 -9151.598} C_VEL
LIN {X 0,Y 439.394,Z 290.752,A -85,B 0,C 180,E1 -9154.415,E2 -9154.415} C_VEL
LIN {X 0,Y 439.36,Z 290.752,A -85,B 0,C 180,E1 -9157.424,E2 -9157.424} C_VEL
LIN {X 0,Y 439.438,Z 290.745,A -85,B 0,C 180,E1 -9160.663,E2 -9160.663} C_VEL
LIN {X 0,Y 439.459,Z 290.738,A -85,B 0,C 180,E1 -9164.225,E2 -9164.225} C_VEL
LIN {X 0,Y 439.48,Z 290.733,A -85,B 0,C 180,E1 -9168.001,E2 -9168.001} C_VEL
LIN {X 0,Y 439.544,Z 290.726,A -85,B 0,C 180,E1 -9171.726,E2 -9171.726} C_VEL
LIN {X 0,Y 439.618,Z 290.724,A -85,B 0,C 180,E1 -9174.496,E2 -9174.496} C_VEL
LIN {X 0,Y 439.633,Z 290.718,A -85,B 0,C 180,E1 -9178.168,E2 -9178.168} C_VEL
LIN {X 0,Y 439.761,Z 290.7,A -85,B 0,C 180,E1 -9180,E2 -9180} C_VEL
LIN {X 0,Y 439.652,Z 290.72,A -85,B 0,C 180,E1 -9182.749,E2 -9182.749} C_VEL
LIN {X 0,Y 439.615,Z 290.72,A -85,B 0,C 180,E1 -9186.426,E2 -9186.426} C_VEL
LIN {X 0,Y 439.497,Z 290.737,A -85,B 0,C 180,E1 -9189.202,E2 -9189.202} C_VEL
LIN {X 0,Y 439.463,Z 290.743,A -85,B 0,C 180,E1 -9192.938,E2 -9192.938} C_VEL
LIN {X 0,Y 439.444,Z 290.742,A -85,B 0,C 180,E1 -9196.349,E2 -9196.349} C_VEL
LIN {X 0,Y 439.399,Z 290.749,A -85,B 0,C 180,E1 -9199.627,E2 -9199.627} C_VEL
LIN {X 0,Y 439.361,Z 290.752,A -85,B 0,C 180,E1 -9202.576,E2 -9202.576} C_VEL
LIN {X 0,Y 439.395,Z 290.75,A -85,B 0,C 180,E1 -9205.586,E2 -9205.586} C_VEL
LIN {X 0,Y 439.415,Z 290.746,A -85,B 0,C 180,E1 -9208.674,E2 -9208.674} C_VEL
LIN {X 0,Y 439.366,Z 290.748,A -85,B 0,C 180,E1 -9212.031,E2 -9212.031} C_VEL
LIN {X 0,Y 439.391,Z 290.751,A -85,B 0,C 180,E1 -9215.341,E2 -9215.341} C_VEL
LIN {X 0,Y 439.362,Z 290.749,A -85,B 0,C 180,E1 -9218.598,E2 -9218.598} C_VEL
LIN {X 0,Y 439.377,Z 290.754,A -85,B 0,C 180,E1 -9221.256,E2 -9221.256} C_VEL
LIN {X 0,Y 439.397,Z 290.75,A -85,B 0,C 180,E1 -9224.731,E2 -9224.731} C_VEL
LIN {X 0,Y 439.357,Z 290.758,A -85,B 0,C 180,E1 -9227.792,E2 -9227.792} C_VEL
LIN {X 0,Y 439.357,Z 290.758,A -85,B 0,C 180,E1 -9231.403,E2 -9231.403} C_VEL
LIN {X 0,Y 439.395,Z 290.747,A -85,B 0,C 180,E1 -9234.844,E2 -9234.844} C_VEL
LIN {X 0,Y 439.372,Z 290.756,A -85,B 0,C 180,E1 -9238.14,E2 -9238.14} C_VEL
LIN {X 0,Y 439.431,Z 290.91,A -85,B 0,C 180,E1 -9240.095,E2 -9240.095} C_VEL
LIN {X 0,Y 440.989,Z 299.347,A -85,B 0,C 180,E1 -9241.957,E2 -9241.957} C_VEL
LIN {X 0,Y 440.956,Z 303.034,A -85,B 0,C 180,E1 -9242.71,E2 -9242.71} C_VEL
LIN {X 0,Y 444.779,Z 320.141,A -85,B 0,C 180,E1 -9243.187,E2 -9243.187} C_VEL
LIN {X 0,Y 443.753,Z 411.03,A -85,B 0,C 180,E1 -9244.7,E2 -9244.7} C_VEL
LIN {X 0,Y 443.448,Z 424.81,A -85,B 0,C 180,E1 -9245.136,E2 -9245.136} C_VEL
LIN {X 0,Y 442.952,Z 436.94,A -85,B 0,C 180,E1 -9245.7,E2 -9245.7} C_VEL
LIN {X 0,Y 442.36,Z 449.129,A -85,B 0,C 180,E1 -9246.474,E2 -9246.474} C_VEL
LIN {X 0,Y 441.767,Z 459.635,A -85,B 0,C 180,E1 -9247.328,E2 -9247.328} C_VEL
LIN {X 0,Y 441.091,Z 470.071,A -85,B 0,C 180,E1 -9248.38,E2 -9248.38} C_VEL
LIN {X 0,Y 440.55,Z 478.711,A -85,B 0,C 180,E1 -9249.455,E2 -9249.455} C_VEL
LIN {X 0,Y 439.983,Z 486.278,A -85,B 0,C 180,E1 -9250.589,E2 -9250.589} C_VEL
LIN {X 0,Y 439.498,Z 493.691,A -85,B 0,C 180,E1 -9251.952,E2 -9251.952} C_VEL
LIN {X 0,Y 438.628,Z 496.817,A -85,B 0,C 180,E1 -9252.601,E2 -9252.601} C_VEL
LIN {X 0,Y 435.471,Z 501.5,A -85,B 0,C 180,E1 -9253.672,E2 -9253.672} C_VEL
LIN {X 0,Y 432.365,Z 505.488,A -85,B 0,C 180,E1 -9254.799,E2 -9254.799} C_VEL
LIN {X 0,Y 431.586,Z 507.493,A -85,B 0,C 180,E1 -9255.528,E2 -9255.528} C_VEL
LIN {X 0,Y 431.422,Z 510.312,A -85,B 0,C 180,E1 -9256.817,E2 -9256.817} C_VEL
LIN {X 0,Y 431.341,Z 512.003,A -85,B 0,C 180,E1 -9257.853,E2 -9257.853} C_VEL
LIN {X 0,Y 431.216,Z 513.706,A -85,B 0,C 180,E1 -9259.673,E2 -9259.673} C_VEL
LIN {X 0,Y 431.218,Z 513.935,A -85,B 0,C 180,E1 -9261.566,E2 -9261.566} C_VEL
LIN {X 0,Y 431.25,Z 513.433,A -85,B 0,C 180,E1 -9262.509,E2 -9262.509} C_VEL
LIN {X 0,Y 431.355,Z 512.273,A -85,B 0,C 180,E1 -9263.655,E2 -9263.655} C_VEL
LIN {X 0,Y 431.353,Z 509.523,A -85,B 0,C 180,E1 -9265.328,E2 -9265.328} C_VEL
LIN {X 0,Y 431.588,Z 506.105,A -85,B 0,C 180,E1 -9266.733,E2 -9266.733} C_VEL
LIN {X 0,Y 431.704,Z 501.634,A -85,B 0,C 180,E1 -9268.135,E2 -9268.135} C_VEL
LIN {X 0,Y 432.196,Z 494.834,A -85,B 0,C 180,E1 -9269.768,E2 -9269.768} C_VEL
LIN {X 0,Y 432.595,Z 487.492,A -85,B 0,C 180,E1 -9271.164,E2 -9271.164} C_VEL
LIN {X 0,Y 433.087,Z 480.006,A -85,B 0,C 180,E1 -9272.326,E2 -9272.326} C_VEL
LIN {X 0,Y 433.554,Z 470.974,A -85,B 0,C 180,E1 -9273.486,E2 -9273.486} C_VEL
LIN {X 0,Y 434.127,Z 460.941,A -85,B 0,C 180,E1 -9274.527,E2 -9274.527} C_VEL
LIN {X 0,Y 434.781,Z 449.802,A -85,B 0,C 180,E1 -9275.45,E2 -9275.45} C_VEL
LIN {X 0,Y 435.263,Z 439.288,A -85,B 0,C 180,E1 -9276.141,E2 -9276.141} C_VEL
LIN {X 0,Y 435.628,Z 426.67,A -85,B 0,C 180,E1 -9276.776,E2 -9276.776} C_VEL
LIN {X 0,Y 435.972,Z 414.003,A -85,B 0,C 180,E1 -9277.207,E2 -9277.207} C_VEL
LIN {X 0,Y 436.215,Z 397.929,A -85,B 0,C 180,E1 -9277.522,E2 -9277.522} C_VEL
LIN {X 0,Y 437.052,Z 320.44,A -85,B 0,C 180,E1 -9278.791,E2 -9278.791} C_VEL
LIN {X 0,Y 433.709,Z 303.131,A -85,B 0,C 180,E1 -9279.215,E2 -9279.215} C_VEL
LIN {X 0,Y 433.357,Z 296.996,A -85,B 0,C 180,E1 -9280.513,E2 -9280.513} C_VEL
LIN {X 0,Y 432.454,Z 291.618,A -85,B 0,C 180,E1 -9281.721,E2 -9281.721} C_VEL
LIN {X 0,Y 432.397,Z 291.622,A -85,B 0,C 180,E1 -9285.074,E2 -9285.074} C_VEL
LIN {X 0,Y 432.362,Z 291.624,A -85,B 0,C 180,E1 -9287.99,E2 -9287.99} C_VEL
LIN {X 0,Y 432.355,Z 291.63,A -85,B 0,C 180,E1 -9290.954,E2 -9290.954} C_VEL
LIN {X 0,Y 432.358,Z 291.627,A -85,B 0,C 180,E1 -9294.454,E2 -9294.454} C_VEL
LIN {X 0,Y 432.305,Z 291.636,A -85,B 0,C 180,E1 -9297.078,E2 -9297.078} C_VEL
LIN {X 0,Y 432.343,Z 291.626,A -85,B 0,C 180,E1 -9300.261,E2 -9300.261} C_VEL
LIN {X 0,Y 432.319,Z 291.631,A -85,B 0,C 180,E1 -9303.555,E2 -9303.555} C_VEL
LIN {X 0,Y 432.342,Z 291.626,A -85,B 0,C 180,E1 -9305.818,E2 -9305.818} C_VEL
LIN {X 0,Y 432.307,Z 291.636,A -85,B 0,C 180,E1 -9309.348,E2 -9309.348} C_VEL
LIN {X 0,Y 432.308,Z 291.631,A -85,B 0,C 180,E1 -9311.801,E2 -9311.801} C_VEL
LIN {X 0,Y 432.339,Z 291.626,A -85,B 0,C 180,E1 -9314.347,E2 -9314.347} C_VEL
LIN {X 0,Y 432.307,Z 291.634,A -85,B 0,C 180,E1 -9317.018,E2 -9317.018} C_VEL
LIN {X 0,Y 432.293,Z 291.635,A -85,B 0,C 180,E1 -9319.828,E2 -9319.828} C_VEL
LIN {X 0,Y 432.304,Z 291.633,A -85,B 0,C 180,E1 -9323.021,E2 -9323.021} C_VEL
LIN {X 0,Y 432.338,Z 291.629,A -85,B 0,C 180,E1 -9326.002,E2 -9326.002} C_VEL
LIN {X 0,Y 432.351,Z 291.631,A -85,B 0,C 180,E1 -9329.49,E2 -9329.49} C_VEL
LIN {X 0,Y 432.347,Z 291.63,A -85,B 0,C 180,E1 -9331.874,E2 -9331.874} C_VEL
LIN {X 0,Y 432.326,Z 291.628,A -85,B 0,C 180,E1 -9334.997,E2 -9334.997} C_VEL
LIN {X 0,Y 432.363,Z 291.628,A -85,B 0,C 180,E1 -9338.046,E2 -9338.046} C_VEL
LIN {X 0,Y 432.389,Z 291.62,A -85,B 0,C 180,E1 -9341.029,E2 -9341.029} C_VEL
LIN {X 0,Y 432.434,Z 291.622,A -85,B 0,C 180,E1 -9343.961,E2 -9343.961} C_VEL
LIN {X 0,Y 432.459,Z 291.616,A -85,B 0,C 180,E1 -9347.803,E2 -9347.803} C_VEL
LIN {X 0,Y 432.451,Z 291.614,A -85,B 0,C 180,E1 -9351.589,E2 -9351.589} C_VEL
LIN {X 0,Y 432.575,Z 291.602,A -85,B 0,C 180,E1 -9354.406,E2 -9354.406} C_VEL
LIN {X 0,Y 432.6,Z 291.6,A -85,B 0,C 180,E1 -9358.138,E2 -9358.138} C_VEL
LIN {X 0,Y 432.524,Z 291.604,A -85,B 0,C 180,E1 -9360.931,E2 -9360.931} C_VEL
LIN {X 0,Y 432.56,Z 291.601,A -85,B 0,C 180,E1 -9362.794,E2 -9362.794} C_VEL
LIN {X 0,Y 432.518,Z 291.611,A -85,B 0,C 180,E1 -9366.531,E2 -9366.531} C_VEL
LIN {X 0,Y 432.422,Z 291.616,A -85,B 0,C 180,E1 -9369.353,E2 -9369.353} C_VEL
LIN {X 0,Y 432.435,Z 291.619,A -85,B 0,C 180,E1 -9372.803,E2 -9372.803} C_VEL
LIN {X 0,Y 432.414,Z 291.623,A -85,B 0,C 180,E1 -9376.477,E2 -9376.477} C_VEL
LIN {X 0,Y 432.341,Z 291.626,A -85,B 0,C 180,E1 -9379.96,E2 -9379.96} C_VEL
LIN {X 0,Y 432.313,Z 291.635,A -85,B 0,C 180,E1 -9382.964,E2 -9382.964} C_VEL
LIN {X 0,Y 432.322,Z 291.628,A -85,B 0,C 180,E1 -9386.035,E2 -9386.035} C_VEL
LIN {X 0,Y 432.324,Z 291.633,A -85,B 0,C 180,E1 -9389.189,E2 -9389.189} C_VEL
LIN {X 0,Y 432.323,Z 291.63,A -85,B 0,C 180,E1 -9392.443,E2 -9392.443} C_VEL
LIN {X 0,Y 432.339,Z 291.627,A -85,B 0,C 180,E1 -9395.818,E2 -9395.818} C_VEL
LIN {X 0,Y 432.305,Z 291.636,A -85,B 0,C 180,E1 -9399.348,E2 -9399.348} C_VEL
LIN {X 0,Y 432.306,Z 291.632,A -85,B 0,C 180,E1 -9401.8,E2 -9401.8} C_VEL
LIN {X 0,Y 432.336,Z 291.626,A -85,B 0,C 180,E1 -9404.347,E2 -9404.347} C_VEL
LIN {X 0,Y 432.305,Z 291.635,A -85,B 0,C 180,E1 -9407.018,E2 -9407.018} C_VEL
LIN {X 0,Y 432.29,Z 291.635,A -85,B 0,C 180,E1 -9409.828,E2 -9409.828} C_VEL
LIN {X 0,Y 432.301,Z 291.634,A -85,B 0,C 180,E1 -9413.021,E2 -9413.021} C_VEL
LIN {X 0,Y 432.336,Z 291.629,A -85,B 0,C 180,E1 -9416.001,E2 -9416.001} C_VEL
LIN {X 0,Y 432.349,Z 291.632,A -85,B 0,C 180,E1 -9419.49,E2 -9419.49} C_VEL
LIN {X 0,Y 432.413,Z 291.823,A -85,B 0,C 180,E1 -9422.733,E2 -9422.733} C_VEL
LIN {X 0,Y 434.988,Z 305.538,A -85,B 0,C 180,E1 -9425.415,E2 -9425.415} C_VEL
LIN {X 0,Y 434.363,Z 319.249,A -85,B 0,C 180,E1 -9427.902,E2 -9427.902} C_VEL
LIN {X 0,Y 433.46,Z 336.975,A -85,B 0,C 180,E1 -9431.078,E2 -9431.078} C_VEL
LIN {X 0,Y 433.263,Z 340.966,A -85,B 0,C 180,E1 -9431.789,E2 -9431.789} C_VEL
LIN {X 0,Y 436.802,Z 367.048,A -85,B 0,C 180,E1 -9432.357,E2 -9432.357} C_VEL
LIN {X 0,Y 435.995,Z 449.793,A -85,B 0,C 180,E1 -9433.735,E2 -9433.735} C_VEL
LIN {X 0,Y 435.458,Z 463.05,A -85,B 0,C 180,E1 -9434.135,E2 -9434.135} C_VEL
LIN {X 0,Y 434.966,Z 475.819,A -85,B 0,C 180,E1 -9434.717,E2 -9434.717} C_VEL
LIN {X 0,Y 434.311,Z 487.941,A -85,B 0,C 180,E1 -9435.473,E2 -9435.473} C_VEL
LIN {X 0,Y 433.741,Z 499.059,A -85,B 0,C 180,E1 -9436.369,E2 -9436.369} C_VEL
LIN {X 0,Y 433.081,Z 509.94,A -85,B 0,C 180,E1 -9437.464,E2 -9437.464} C_VEL
LIN {X 0,Y 432.582,Z 518.454,A -85,B 0,C 180,E1 -9438.52,E2 -9438.52} C_VEL
LIN {X 0,Y 432.006,Z 527.67,A -85,B 0,C 180,E1 -9439.927,E2 -9439.927} C_VEL
LIN {X 0,Y 431.673,Z 535.095,A -85,B 0,C 180,E1 -9441.338,E2 -9441.338} C_VEL
LIN {X 0,Y 431.411,Z 541.905,A -85,B 0,C 180,E1 -9442.981,E2 -9442.981} C_VEL
LIN {X 0,Y 431.288,Z 546.393,A -85,B 0,C 180,E1 -9444.389,E2 -9444.389} C_VEL
LIN {X 0,Y 431.276,Z 548.761,A -85,B 0,C 180,E1 -9445.326,E2 -9445.326} C_VEL
LIN {X 0,Y 431.199,Z 550.69,A -85,B 0,C 180,E1 -9446.261,E2 -9446.261} C_VEL
LIN {X 0,Y 431.279,Z 552.19,A -85,B 0,C 180,E1 -9447.197,E2 -9447.197} C_VEL
LIN {X 0,Y 431.24,Z 553.235,A -85,B 0,C 180,E1 -9448.132,E2 -9448.132} C_VEL
LIN {X 0,Y 431.223,Z 554.155,A -85,B 0,C 180,E1 -9449.999,E2 -9449.999} C_VEL
LIN {X 0,Y 431.22,Z 554.019,A -85,B 0,C 180,E1 -9450.933,E2 -9450.933} C_VEL
LIN {X 0,Y 431.28,Z 552.496,A -85,B 0,C 180,E1 -9452.802,E2 -9452.802} C_VEL
LIN {X 0,Y 431.197,Z 551.14,A -85,B 0,C 180,E1 -9453.737,E2 -9453.737} C_VEL
LIN {X 0,Y 431.293,Z 548.287,A -85,B 0,C 180,E1 -9455.141,E2 -9455.141} C_VEL
LIN {X 0,Y 431.375,Z 544.408,A -85,B 0,C 180,E1 -9456.548,E2 -9456.548} C_VEL
LIN {X 0,Y 431.558,Z 539.409,A -85,B 0,C 180,E1 -9457.956,E2 -9457.956} C_VEL
LIN {X 0,Y 431.88,Z 533.143,A -85,B 0,C 180,E1 -9459.365,E2 -9459.365} C_VEL
LIN {X 0,Y 432.343,Z 525.335,A -85,B 0,C 180,E1 -9460.774,E2 -9460.774} C_VEL
LIN {X 0,Y 433.091,Z 515.599,A -85,B 0,C 180,E1 -9462.178,E2 -9462.178} C_VEL
LIN {X 0,Y 433.741,Z 505.243,A -85,B 0,C 180,E1 -9463.381,E2 -9463.381} C_VEL
LIN {X 0,Y 434.474,Z 494.19,A -85,B 0,C 180,E1 -9464.4,E2 -9464.4} C_VEL
LIN {X 0,Y 435.156,Z 483.078,A -85,B 0,C 180,E1 -9465.215,E2 -9465.215} C_VEL
LIN {X 0,Y 435.921,Z 470.723,A -85,B 0,C 180,E1 -9465.906,E2 -9465.906} C_VEL
LIN {X 0,Y 436.508,Z 457.592,A -85,B 0,C 180,E1 -9466.425,E2 -9466.425} C_VEL
LIN {X 0,Y 436.921,Z 444.957,A -85,B 0,C 180,E1 -9466.739,E2 -9466.739} C_VEL
LIN {X 0,Y 437.695,Z 365.814,A -85,B 0,C 180,E1 -9468.062,E2 -9468.062} C_VEL
LIN {X 0,Y 434.071,Z 342.968,A -85,B 0,C 180,E1 -9468.632,E2 -9468.632} C_VEL
LIN {X 0,Y 433.63,Z 340.535,A -85,B 0,C 180,E1 -9468.713,E2 -9468.713} C_VEL
LIN {X 0,Y 434.747,Z 322.046,A -85,B 0,C 180,E1 -9472.076,E2 -9472.076} C_VEL
LIN {X 0,Y 435.534,Z 307.316,A -85,B 0,C 180,E1 -9474.805,E2 -9474.805} C_VEL
LIN {X 0,Y 433.464,Z 296.567,A -85,B 0,C 180,E1 -9476.999,E2 -9476.999} C_VEL
LIN {X 0,Y 432.394,Z 291.63,A -85,B 0,C 180,E1 -9478.056,E2 -9478.056} C_VEL
LIN {X 0,Y 432.319,Z 291.638,A -85,B 0,C 180,E1 -9481.346,E2 -9481.346} C_VEL
LIN {X 0,Y 432.335,Z 291.636,A -85,B 0,C 180,E1 -9484.677,E2 -9484.677} C_VEL
LIN {X 0,Y 432.33,Z 291.634,A -85,B 0,C 180,E1 -9488.15,E2 -9488.15} C_VEL
LIN {X 0,Y 432.33,Z 291.627,A -85,B 0,C 180,E1 -9491.601,E2 -9491.601} C_VEL
LIN {X 0,Y 432.331,Z 291.635,A -85,B 0,C 180,E1 -9494.347,E2 -9494.347} C_VEL
LIN {X 0,Y 432.317,Z 291.632,A -85,B 0,C 180,E1 -9497.015,E2 -9497.015} C_VEL
LIN {X 0,Y 432.338,Z 291.627,A -85,B 0,C 180,E1 -9499.819,E2 -9499.819} C_VEL
LIN {X 0,Y 432.303,Z 291.634,A -85,B 0,C 180,E1 -9503.022,E2 -9503.022} C_VEL
LIN {X 0,Y 432.354,Z 291.624,A -85,B 0,C 180,E1 -9505.997,E2 -9505.997} C_VEL
LIN {X 0,Y 432.344,Z 291.625,A -85,B 0,C 180,E1 -9509.489,E2 -9509.489} C_VEL
LIN {X 0,Y 432.387,Z 291.624,A -85,B 0,C 180,E1 -9512.928,E2 -9512.928} C_VEL
LIN {X 0,Y 432.364,Z 291.62,A -85,B 0,C 180,E1 -9516.023,E2 -9516.023} C_VEL
LIN {X 0,Y 432.347,Z 291.624,A -85,B 0,C 180,E1 -9519.046,E2 -9519.046} C_VEL
LIN {X 0,Y 432.375,Z 291.623,A -85,B 0,C 180,E1 -9522.011,E2 -9522.011} C_VEL
LIN {X 0,Y 432.393,Z 291.627,A -85,B 0,C 180,E1 -9524.927,E2 -9524.927} C_VEL
LIN {X 0,Y 432.456,Z 291.608,A -85,B 0,C 180,E1 -9527.803,E2 -9527.803} C_VEL
LIN {X 0,Y 432.488,Z 291.605,A -85,B 0,C 180,E1 -9531.59,E2 -9531.59} C_VEL
LIN {X 0,Y 432.594,Z 291.598,A -85,B 0,C 180,E1 -9534.406,E2 -9534.406} C_VEL
LIN {X 0,Y 432.603,Z 291.594,A -85,B 0,C 180,E1 -9538.138,E2 -9538.138} C_VEL
LIN {X 0,Y 432.731,Z 291.576,A -85,B 0,C 180,E1 -9540,E2 -9540} C_VEL
LIN {X 0,Y 432.601,Z 291.599,A -85,B 0,C 180,E1 -9542.794,E2 -9542.794} C_VEL
LIN {X 0,Y 432.57,Z 291.599,A -85,B 0,C 180,E1 -9546.531,E2 -9546.531} C_VEL
LIN {X 0,Y 432.44,Z 291.616,A -85,B 0,C 180,E1 -9549.353,E2 -9549.353} C_VEL
LIN {X 0,Y 432.428,Z 291.62,A -85,B 0,C 180,E1 -9552.804,E2 -9552.804} C_VEL
LIN {X 0,Y 432.409,Z 291.619,A -85,B 0,C 180,E1 -9556.479,E2 -9556.479} C_VEL
LIN {X 0,Y 432.336,Z 291.628,A -85,B 0,C 180,E1 -9559.961,E2 -9559.961} C_VEL
LIN {X 0,Y 432.315,Z 291.634,A -85,B 0,C 180,E1 -9562.965,E2 -9562.965} C_VEL
LIN {X 0,Y 432.358,Z 291.624,A -85,B 0,C 180,E1 -9566.033,E2 -9566.033} C_VEL
LIN {X 0,Y 432.34,Z 291.63,A -85,B 0,C 180,E1 -9569.188,E2 -9569.188} C_VEL
LIN {X 0,Y 432.32,Z 291.626,A -85,B 0,C 180,E1 -9572.444,E2 -9572.444} C_VEL
LIN {X 0,Y 432.341,Z 291.629,A -85,B 0,C 180,E1 -9575.632,E2 -9575.632} C_VEL
LIN {X 0,Y 432.325,Z 291.626,A -85,B 0,C 180,E1 -9578.713,E2 -9578.713} C_VEL
LIN {X 0,Y 432.312,Z 291.634,A -85,B 0,C 180,E1 -9581.8,E2 -9581.8} C_VEL
LIN {X 0,Y 432.333,Z 291.629,A -85,B 0,C 180,E1 -9584.348,E2 -9584.348} C_VEL
LIN {X 0,Y 432.306,Z 291.636,A -85,B 0,C 180,E1 -9587.019,E2 -9587.019} C_VEL
LIN {X 0,Y 432.288,Z 291.639,A -85,B 0,C 180,E1 -9589.829,E2 -9589.829} C_VEL
LIN {X 0,Y 432.299,Z 291.636,A -85,B 0,C 180,E1 -9593.022,E2 -9593.022} C_VEL
LIN {X 0,Y 432.358,Z 291.629,A -85,B 0,C 180,E1 -9595.998,E2 -9595.998} C_VEL
LIN {X 0,Y 432.345,Z 291.633,A -85,B 0,C 180,E1 -9599.491,E2 -9599.491} C_VEL
LIN {X 0,Y 432.353,Z 291.757,A -85,B 0,C 180,E1 -9599.809,E2 -9599.809} C_VEL
LIN {X 0,Y 434.049,Z 300.363,A -85,B 0,C 180,E1 -9601.747,E2 -9601.747} C_VEL
LIN {X 0,Y 434.151,Z 303.553,A -85,B 0,C 180,E1 -9602.375,E2 -9602.375} C_VEL
LIN {X 0,Y 438.176,Z 321.434,A -85,B 0,C 180,E1 -9602.888,E2 -9602.888} C_VEL
LIN {X 0,Y 437.025,Z 410.955,A -85,B 0,C 180,E1 -9604.394,E2 -9604.394} C_VEL
LIN {X 0,Y 436.75,Z 424.488,A -85,B 0,C 180,E1 -9604.823,E2 -9604.823} C_VEL
LIN {X 0,Y 436.186,Z 437.355,A -85,B 0,C 180,E1 -9605.425,E2 -9605.425} C_VEL
LIN {X 0,Y 435.562,Z 449.518,A -85,B 0,C 180,E1 -9606.211,E2 -9606.211} C_VEL
LIN {X 0,Y 434.878,Z 461.125,A -85,B 0,C 180,E1 -9607.179,E2 -9607.179} C_VEL
LIN {X 0,Y 434.159,Z 471.473,A -85,B 0,C 180,E1 -9608.267,E2 -9608.267} C_VEL
LIN {X 0,Y 433.465,Z 481.568,A -85,B 0,C 180,E1 -9609.599,E2 -9609.599} C_VEL
LIN {X 0,Y 432.867,Z 489.285,A -85,B 0,C 180,E1 -9610.854,E2 -9610.854} C_VEL
LIN {X 0,Y 432.325,Z 496.292,A -85,B 0,C 180,E1 -9612.254,E2 -9612.254} C_VEL
LIN {X 0,Y 431.955,Z 502.126,A -85,B 0,C 180,E1 -9613.73,E2 -9613.73} C_VEL
LIN {X 0,Y 431.607,Z 507.131,A -85,B 0,C 180,E1 -9615.382,E2 -9615.382} C_VEL
LIN {X 0,Y 431.586,Z 507.493,A -85,B 0,C 180,E1 -9615.528,E2 -9615.528} C_VEL
LIN {X 0,Y 430.833,Z 509.289,A -85,B 0,C 180,E1 -9616.271,E2 -9616.271} C_VEL
LIN {X 0,Y 427.851,Z 511.78,A -85,B 0,C 180,E1 -9617.489,E2 -9617.489} C_VEL
LIN {X 0,Y 425.345,Z 513.214,A -85,B 0,C 180,E1 -9618.488,E2 -9618.488} C_VEL
LIN {X 0,Y 424.235,Z 513.871,A -85,B 0,C 180,E1 -9619.27,E2 -9619.27} C_VEL
LIN {X 0,Y 424.126,Z 513.994,A -85,B 0,C 180,E1 -9619.536,E2 -9619.536} C_VEL
LIN {X 0,Y 424.122,Z 514.286,A -85,B 0,C 180,E1 -9621.424,E2 -9621.424} C_VEL
LIN {X 0,Y 424.162,Z 513.855,A -85,B 0,C 180,E1 -9622.383,E2 -9622.383} C_VEL
LIN {X 0,Y 424.263,Z 512.585,A -85,B 0,C 180,E1 -9623.68,E2 -9623.68} C_VEL
LIN {X 0,Y 424.273,Z 510.07,A -85,B 0,C 180,E1 -9625.25,E2 -9625.25} C_VEL
LIN {X 0,Y 424.502,Z 506.734,A -85,B 0,C 180,E1 -9626.679,E2 -9626.679} C_VEL
LIN {X 0,Y 424.632,Z 502.351,A -85,B 0,C 180,E1 -9628.104,E2 -9628.104} C_VEL
LIN {X 0,Y 425,Z 496.774,A -85,B 0,C 180,E1 -9629.527,E2 -9629.527} C_VEL
LIN {X 0,Y 425.445,Z 489.809,A -85,B 0,C 180,E1 -9630.947,E2 -9630.947} C_VEL
LIN {X 0,Y 426.039,Z 481.109,A -85,B 0,C 180,E1 -9632.364,E2 -9632.364} C_VEL
LIN {X 0,Y 426.539,Z 472.226,A -85,B 0,C 180,E1 -9633.543,E2 -9633.543} C_VEL
LIN {X 0,Y 427.119,Z 462.455,A -85,B 0,C 180,E1 -9634.602,E2 -9634.602} C_VEL
LIN {X 0,Y 427.779,Z 451.624,A -85,B 0,C 180,E1 -9635.539,E2 -9635.539} C_VEL
LIN {X 0,Y 428.364,Z 439.524,A -85,B 0,C 180,E1 -9636.359,E2 -9636.359} C_VEL
LIN {X 0,Y 428.762,Z 426.86,A -85,B 0,C 180,E1 -9637.003,E2 -9637.003} C_VEL
LIN {X 0,Y 429.116,Z 414.106,A -85,B 0,C 180,E1 -9637.441,E2 -9637.441} C_VEL
LIN {X 0,Y 429.387,Z 396.15,A -85,B 0,C 180,E1 -9637.791,E2 -9637.791} C_VEL
LIN {X 0,Y 430.247,Z 321.594,A -85,B 0,C 180,E1 -9639.029,E2 -9639.029} C_VEL
LIN {X 0,Y 426.78,Z 303.439,A -85,B 0,C 180,E1 -9639.479,E2 -9639.479} C_VEL
LIN {X 0,Y 426.321,Z 297.826,A -85,B 0,C 180,E1 -9640.688,E2 -9640.688} C_VEL
LIN {X 0,Y 425.434,Z 292.493,A -85,B 0,C 180,E1 -9641.918,E2 -9641.918} C_VEL
LIN {X 0,Y 425.351,Z 292.498,A -85,B 0,C 180,E1 -9645.33,E2 -9645.33} C_VEL
LIN {X 0,Y 425.325,Z 292.503,A -85,B 0,C 180,E1 -9648.298,E2 -9648.298} C_VEL
LIN {X 0,Y 425.298,Z 292.505,A -85,B 0,C 180,E1 -9651.319,E2 -9651.319} C_VEL
LIN {X 0,Y 425.305,Z 292.508,A -85,B 0,C 180,E1 -9654.651,E2 -9654.651} C_VEL
LIN {X 0,Y 425.251,Z 292.51,A -85,B 0,C 180,E1 -9657.565,E2 -9657.565} C_VEL
LIN {X 0,Y 425.294,Z 292.509,A -85,B 0,C 180,E1 -9660.761,E2 -9660.761} C_VEL
LIN {X 0,Y 425.297,Z 292.504,A -85,B 0,C 180,E1 -9664.284,E2 -9664.284} C_VEL
LIN {X 0,Y 425.281,Z 292.507,A -85,B 0,C 180,E1 -9667.695,E2 -9667.695} C_VEL
LIN {X 0,Y 425.249,Z 292.51,A -85,B 0,C 180,E1 -9670.514,E2 -9670.514} C_VEL
LIN {X 0,Y 425.252,Z 292.516,A -85,B 0,C 180,E1 -9673.349,E2 -9673.349} C_VEL
LIN {X 0,Y 425.262,Z 292.508,A -85,B 0,C 180,E1 -9676.043,E2 -9676.043} C_VEL
LIN {X 0,Y 425.252,Z 292.509,A -85,B 0,C 180,E1 -9678.618,E2 -9678.618} C_VEL
LIN {X 0,Y 425.283,Z 292.509,A -85,B 0,C 180,E1 -9681.099,E2 -9681.099} C_VEL
LIN {X 0,Y 425.299,Z 292.503,A -85,B 0,C 180,E1 -9684.664,E2 -9684.664} C_VEL
LIN {X 0,Y 425.268,Z 292.509,A -85,B 0,C 180,E1 -9688.073,E2 -9688.073} C_VEL
LIN {X 0,Y 425.315,Z 292.505,A -85,B 0,C 180,E1 -9691.366,E2 -9691.366} C_VEL
LIN {X 0,Y 425.264,Z 292.508,A -85,B 0,C 180,E1 -9694.552,E2 -9694.552} C_VEL
LIN {X 0,Y 425.297,Z 292.511,A -85,B 0,C 180,E1 -9697.73,E2 -9697.73} C_VEL
LIN {X 0,Y 425.366,Z 292.495,A -85,B 0,C 180,E1 -9700.704,E2 -9700.704} C_VEL
LIN {X 0,Y 425.392,Z 292.496,A -85,B 0,C 180,E1 -9703.688,E2 -9703.688} C_VEL
LIN {X 0,Y 425.414,Z 292.492,A -85,B 0,C 180,E1 -9707.598,E2 -9707.598} C_VEL
LIN {X 0,Y 425.4,Z 292.492,A -85,B 0,C 180,E1 -9711.449,E2 -9711.449} C_VEL
LIN {X 0,Y 425.53,Z 292.48,A -85,B 0,C 180,E1 -9714.313,E2 -9714.313} C_VEL
LIN {X 0,Y 425.569,Z 292.476,A -85,B 0,C 180,E1 -9718.107,E2 -9718.107} C_VEL
LIN {X 0,Y 425.489,Z 292.48,A -85,B 0,C 180,E1 -9720.946,E2 -9720.946} C_VEL
LIN {X 0,Y 425.515,Z 292.478,A -85,B 0,C 180,E1 -9722.84,E2 -9722.84} C_VEL
LIN {X 0,Y 425.513,Z 292.477,A -85,B 0,C 180,E1 -9725.687,E2 -9725.687} C_VEL
LIN {X 0,Y 425.397,Z 292.498,A -85,B 0,C 180,E1 -9728.551,E2 -9728.551} C_VEL
LIN {X 0,Y 425.413,Z 292.495,A -85,B 0,C 180,E1 -9732.402,E2 -9732.402} C_VEL
LIN {X 0,Y 425.388,Z 292.496,A -85,B 0,C 180,E1 -9736.312,E2 -9736.312} C_VEL
LIN {X 0,Y 425.332,Z 292.499,A -85,B 0,C 180,E1 -9739.635,E2 -9739.635} C_VEL
LIN {X 0,Y 425.291,Z 292.507,A -85,B 0,C 180,E1 -9742.338,E2 -9742.338} C_VEL
LIN {X 0,Y 425.264,Z 292.509,A -85,B 0,C 180,E1 -9745.447,E2 -9745.447} C_VEL
LIN {X 0,Y 425.302,Z 292.51,A -85,B 0,C 180,E1 -9748.858,E2 -9748.858} C_VEL
LIN {X 0,Y 425.263,Z 292.508,A -85,B 0,C 180,E1 -9751.927,E2 -9751.927} C_VEL
LIN {X 0,Y 425.298,Z 292.508,A -85,B 0,C 180,E1 -9755.336,E2 -9755.336} C_VEL
LIN {X 0,Y 425.283,Z 292.51,A -85,B 0,C 180,E1 -9758.9,E2 -9758.9} C_VEL
LIN {X 0,Y 425.259,Z 292.51,A -85,B 0,C 180,E1 -9762.655,E2 -9762.655} C_VEL
LIN {X 0,Y 425.287,Z 292.513,A -85,B 0,C 180,E1 -9765.283,E2 -9765.283} C_VEL
LIN {X 0,Y 425.25,Z 292.51,A -85,B 0,C 180,E1 -9768.618,E2 -9768.618} C_VEL
LIN {X 0,Y 425.28,Z 292.509,A -85,B 0,C 180,E1 -9771.099,E2 -9771.099} C_VEL
LIN {X 0,Y 425.297,Z 292.504,A -85,B 0,C 180,E1 -9774.663,E2 -9774.663} C_VEL
LIN {X 0,Y 425.266,Z 292.512,A -85,B 0,C 180,E1 -9778.072,E2 -9778.072} C_VEL
LIN {X 0,Y 425.313,Z 292.508,A -85,B 0,C 180,E1 -9781.366,E2 -9781.366} C_VEL
LIN {X 0,Y 425.362,Z 292.628,A -85,B 0,C 180,E1 -9782.514,E2 -9782.514} C_VEL
LIN {X 0,Y 427.96,Z 306.331,A -85,B 0,C 180,E1 -9785.243,E2 -9785.243} C_VEL
LIN {X 0,Y 427.617,Z 316.346,A -85,B 0,C 180,E1 -9787.098,E2 -9787.098} C_VEL
LIN {X 0,Y 426.624,Z 335.094,A -85,B 0,C 180,E1 -9790.518,E2 -9790.518} C_VEL
LIN {X 0,Y 426.289,Z 340.628,A -85,B 0,C 180,E1 -9791.519,E2 -9791.519} C_VEL
LIN {X 0,Y 429.967,Z 366.699,A -85,B 0,C 180,E1 -9792.104,E2 -9792.104} C_VEL
LIN {X 0,Y 429.119,Z 449.233,A -85,B 0,C 180,E1 -9793.497,E2 -9793.497} C_VEL
LIN {X 0,Y 428.595,Z 462.575,A -85,B 0,C 180,E1 -9793.905,E2 -9793.905} C_VEL
LIN {X 0,Y 428.078,Z 474.813,A -85,B 0,C 180,E1 -9794.465,E2 -9794.465} C_VEL
LIN {X 0,Y 427.378,Z 487.139,A -85,B 0,C 180,E1 -9795.232,E2 -9795.232} C_VEL
LIN {X 0,Y 426.768,Z 498.964,A -85,B 0,C 180,E1 -9796.199,E2 -9796.199} C_VEL
LIN {X 0,Y 426.125,Z 509.299,A -85,B 0,C 180,E1 -9797.256,E2 -9797.256} C_VEL
LIN {X 0,Y 425.584,Z 517.87,A -85,B 0,C 180,E1 -9798.328,E2 -9798.328} C_VEL
LIN {X 0,Y 424.948,Z 527.144,A -85,B 0,C 180,E1 -9799.758,E2 -9799.758} C_VEL
LIN {X 0,Y 424.621,Z 534.607,A -85,B 0,C 180,E1 -9801.193,E2 -9801.193} C_VEL
LIN {X 0,Y 424.334,Z 541.462,A -85,B 0,C 180,E1 -9802.864,E2 -9802.864} C_VEL
LIN {X 0,Y 424.195,Z 545.976,A -85,B 0,C 180,E1 -9804.294,E2 -9804.294} C_VEL
LIN {X 0,Y 424.207,Z 548.359,A -85,B 0,C 180,E1 -9805.248,E2 -9805.248} C_VEL
LIN {X 0,Y 424.109,Z 550.299,A -85,B 0,C 180,E1 -9806.199,E2 -9806.199} C_VEL
LIN {X 0,Y 424.19,Z 551.82,A -85,B 0,C 180,E1 -9807.15,E2 -9807.15} C_VEL
LIN {X 0,Y 424.165,Z 552.879,A -85,B 0,C 180,E1 -9808.1,E2 -9808.1} C_VEL
LIN {X 0,Y 424.137,Z 553.819,A -85,B 0,C 180,E1 -9809.999,E2 -9809.999} C_VEL
LIN {X 0,Y 424.136,Z 553.701,A -85,B 0,C 180,E1 -9810.949,E2 -9810.949} C_VEL
LIN {X 0,Y 424.165,Z 553.149,A -85,B 0,C 180,E1 -9811.898,E2 -9811.898} C_VEL
LIN {X 0,Y 424.175,Z 552.202,A -85,B 0,C 180,E1 -9812.849,E2 -9812.849} C_VEL
LIN {X 0,Y 424.108,Z 550.857,A -85,B 0,C 180,E1 -9813.8,E2 -9813.8} C_VEL
LIN {X 0,Y 424.204,Z 548.027,A -85,B 0,C 180,E1 -9815.228,E2 -9815.228} C_VEL
LIN {X 0,Y 424.298,Z 544.174,A -85,B 0,C 180,E1 -9816.658,E2 -9816.658} C_VEL
LIN {X 0,Y 424.504,Z 539.203,A -85,B 0,C 180,E1 -9818.089,E2 -9818.089} C_VEL
LIN {X 0,Y 424.824,Z 532.968,A -85,B 0,C 180,E1 -9819.522,E2 -9819.522} C_VEL
LIN {X 0,Y 425.343,Z 525.217,A -85,B 0,C 180,E1 -9820.953,E2 -9820.953} C_VEL
LIN {X 0,Y 426.129,Z 515.527,A -85,B 0,C 180,E1 -9822.38,E2 -9822.38} C_VEL
LIN {X 0,Y 426.77,Z 505.969,A -85,B 0,C 180,E1 -9823.524,E2 -9823.524} C_VEL
LIN {X 0,Y 427.509,Z 495.709,A -85,B 0,C 180,E1 -9824.518,E2 -9824.518} C_VEL
LIN {X 0,Y 428.332,Z 483.282,A -85,B 0,C 180,E1 -9825.463,E2 -9825.463} C_VEL
LIN {X 0,Y 429.117,Z 471.103,A -85,B 0,C 180,E1 -9826.165,E2 -9826.165} C_VEL
LIN {X 0,Y 429.75,Z 458.377,A -85,B 0,C 180,E1 -9826.69,E2 -9826.69} C_VEL
LIN {X 0,Y 430.194,Z 444.979,A -85,B 0,C 180,E1 -9827.039,E2 -9827.039} C_VEL
LIN {X 0,Y 431.047,Z 366.741,A -85,B 0,C 180,E1 -9828.367,E2 -9828.367} C_VEL
LIN {X 0,Y 427.492,Z 344.458,A -85,B 0,C 180,E1 -9828.937,E2 -9828.937} C_VEL
LIN {X 0,Y 426.732,Z 340.277,A -85,B 0,C 180,E1 -9829.052,E2 -9829.052} C_VEL
LIN {X 0,Y 427.902,Z 321.968,A -85,B 0,C 180,E1 -9832.442,E2 -9832.442} C_VEL
LIN {X 0,Y 428.68,Z 309.894,A -85,B 0,C 180,E1 -9834.711,E2 -9834.711} C_VEL
LIN {X 0,Y 427.629,Z 303.103,A -85,B 0,C 180,E1 -9836.095,E2 -9836.095} C_VEL
LIN {X 0,Y 425.343,Z 292.51,A -85,B 0,C 180,E1 -9838.361,E2 -9838.361} C_VEL
LIN {X 0,Y 425.262,Z 292.514,A -85,B 0,C 180,E1 -9841.926,E2 -9841.926} C_VEL
LIN {X 0,Y 425.295,Z 292.51,A -85,B 0,C 180,E1 -9845.336,E2 -9845.336} C_VEL
LIN {X 0,Y 425.289,Z 292.507,A -85,B 0,C 180,E1 -9848.899,E2 -9848.899} C_VEL
LIN {X 0,Y 425.287,Z 292.507,A -85,B 0,C 180,E1 -9851.958,E2 -9851.958} C_VEL
LIN {X 0,Y 425.282,Z 292.507,A -85,B 0,C 180,E1 -9855.283,E2 -9855.283} C_VEL
LIN {X 0,Y 425.272,Z 292.51,A -85,B 0,C 180,E1 -9858.621,E2 -9858.621} C_VEL
LIN {X 0,Y 425.309,Z 292.503,A -85,B 0,C 180,E1 -9861.103,E2 -9861.103} C_VEL
LIN {X 0,Y 425.294,Z 292.506,A -85,B 0,C 180,E1 -9864.664,E2 -9864.664} C_VEL
LIN {X 0,Y 425.261,Z 292.509,A -85,B 0,C 180,E1 -9868.073,E2 -9868.073} C_VEL
LIN {X 0,Y 425.328,Z 292.497,A -85,B 0,C 180,E1 -9871.368,E2 -9871.368} C_VEL
LIN {X 0,Y 425.288,Z 292.511,A -85,B 0,C 180,E1 -9874.554,E2 -9874.554} C_VEL
LIN {X 0,Y 425.284,Z 292.505,A -85,B 0,C 180,E1 -9877.661,E2 -9877.661} C_VEL
LIN {X 0,Y 425.359,Z 292.499,A -85,B 0,C 180,E1 -9880.704,E2 -9880.704} C_VEL
LIN {X 0,Y 425.385,Z 292.489,A -85,B 0,C 180,E1 -9883.688,E2 -9883.688} C_VEL
LIN {X 0,Y 425.408,Z 292.486,A -85,B 0,C 180,E1 -9887.598,E2 -9887.598} C_VEL
LIN {X 0,Y 425.439,Z 292.484,A -85,B 0,C 180,E1 -9891.45,E2 -9891.45} C_VEL
LIN {X 0,Y 425.551,Z 292.474,A -85,B 0,C 180,E1 -9894.313,E2 -9894.313} C_VEL
LIN {X 0,Y 425.572,Z 292.47,A -85,B 0,C 180,E1 -9898.107,E2 -9898.107} C_VEL
LIN {X 0,Y 425.7,Z 292.451,A -85,B 0,C 180,E1 -9900,E2 -9900} C_VEL
LIN {X 0,Y 425.553,Z 292.478,A -85,B 0,C 180,E1 -9902.84,E2 -9902.84} C_VEL
LIN {X 0,Y 425.528,Z 292.477,A -85,B 0,C 180,E1 -9906.639,E2 -9906.639} C_VEL
LIN {X 0,Y 425.398,Z 292.492,A -85,B 0,C 180,E1 -9909.51,E2 -9909.51} C_VEL
LIN {X 0,Y 425.39,Z 292.495,A -85,B 0,C 180,E1 -9912.904,E2 -9912.904} C_VEL
LIN {X 0,Y 425.358,Z 292.498,A -85,B 0,C 180,E1 -9916.605,E2 -9916.605} C_VEL
LIN {X 0,Y 425.325,Z 292.503,A -85,B 0,C 180,E1 -9919.636,E2 -9919.636} C_VEL
LIN {X 0,Y 425.302,Z 292.509,A -85,B 0,C 180,E1 -9923.366,E2 -9923.366} C_VEL
LIN {X 0,Y 425.344,Z 292.501,A -85,B 0,C 180,E1 -9926.845,E2 -9926.845} C_VEL
LIN {X 0,Y 425.289,Z 292.507,A -85,B 0,C 180,E1 -9929.72,E2 -9929.72} C_VEL
LIN {X 0,Y 425.28,Z 292.507,A -85,B 0,C 180,E1 -9933.049,E2 -9933.049} C_VEL
LIN {X 0,Y 425.28,Z 292.506,A -85,B 0,C 180,E1 -9935.929,E2 -9935.929} C_VEL
LIN {X 0,Y 425.261,Z 292.509,A -85,B 0,C 180,E1 -9939.038,E2 -9939.038} C_VEL
LIN {X 0,Y 425.271,Z 292.51,A -85,B 0,C 180,E1 -9941.956,E2 -9941.956} C_VEL
LIN {X 0,Y 425.284,Z 292.512,A -85,B 0,C 180,E1 -9945.284,E2 -9945.284} C_VEL
LIN {X 0,Y 425.25,Z 292.512,A -85,B 0,C 180,E1 -9948.619,E2 -9948.619} C_VEL
LIN {X 0,Y 425.277,Z 292.512,A -85,B 0,C 180,E1 -9951.1,E2 -9951.1} C_VEL
LIN {X 0,Y 425.297,Z 292.503,A -85,B 0,C 180,E1 -9954.665,E2 -9954.665} C_VEL
LIN {X 0,Y 425.265,Z 292.514,A -85,B 0,C 180,E1 -9958.074,E2 -9958.074} C_VEL
LIN {X 0,Y 425.338,Z 292.688,A -85,B 0,C 180,E1 -9959.533,E2 -9959.533} C_VEL
LIN {X 0,Y 427.11,Z 301.254,A -85,B 0,C 180,E1 -9961.499,E2 -9961.499} C_VEL
LIN {X 0,Y 427.216,Z 303.593,A -85,B 0,C 180,E1 -9962.005,E2 -9962.005} C_VEL
LIN {X 0,Y 431.44,Z 321.873,A -85,B 0,C 180,E1 -9962.556,E2 -9962.556} C_VEL
LIN {X 0,Y 430.327,Z 411.029,A -85,B 0,C 180,E1 -9964.082,E2 -9964.082} C_VEL
LIN {X 0,Y 430.027,Z 424.24,A -85,B 0,C 180,E1 -9964.501,E2 -9964.501} C_VEL
LIN {X 0,Y 429.495,Z 436.67,A -85,B 0,C 180,E1 -9965.08,E2 -9965.08} C_VEL
LIN {X 0,Y 428.89,Z 448.312,A -85,B 0,C 180,E1 -9965.817,E2 -9965.817} C_VEL
LIN {X 0,Y 428.143,Z 460.197,A -85,B 0,C 180,E1 -9966.799,E2 -9966.799} C_VEL
LIN {X 0,Y 427.371,Z 470.817,A -85,B 0,C 180,E1 -9967.904,E2 -9967.904} C_VEL
LIN {X 0,Y 426.747,Z 479.436,A -85,B 0,C 180,E1 -9969.011,E2 -9969.011} C_VEL
LIN {X 0,Y 426.016,Z 488.155,A -85,B 0,C 180,E1 -9970.388,E2 -9970.388} C_VEL
LIN {X 0,Y 425.394,Z 496.09,A -85,B 0,C 180,E1 -9971.955,E2 -9971.955} C_VEL
LIN {X 0,Y 425.039,Z 501.237,A -85,B 0,C 180,E1 -9973.23,E2 -9973.23} C_VEL
LIN {X 0,Y 424.687,Z 505.836,A -85,B 0,C 180,E1 -9974.647,E2 -9974.647} C_VEL
LIN {X 0,Y 424.433,Z 509.461,A -85,B 0,C 180,E1 -9976.108,E2 -9976.108} C_VEL
LIN {X 0,Y 424.263,Z 512.36,A -85,B 0,C 180,E1 -9977.784,E2 -9977.784} C_VEL
LIN {X 0,Y 424.126,Z 513.994,A -85,B 0,C 180,E1 -9979.536,E2 -9979.536} C_VEL
LIN {X 0,Y 423.424,Z 514.349,A -85,B 0,C 180,E1 -9980.329,E2 -9980.329} C_VEL
LIN {X 0,Y 420.613,Z 514.404,A -85,B 0,C 180,E1 -9981.621,E2 -9981.621} C_VEL
LIN {X 0,Y 418.269,Z 513.957,A -85,B 0,C 180,E1 -9982.66,E2 -9982.66} C_VEL
LIN {X 0,Y 417.264,Z 513.205,A -85,B 0,C 180,E1 -9983.456,E2 -9983.456} C_VEL
LIN {X 0,Y 417.181,Z 512.868,A -85,B 0,C 180,E1 -9983.724,E2 -9983.724} C_VEL
LIN {X 0,Y 417.215,Z 509.645,A -85,B 0,C 180,E1 -9985.653,E2 -9985.653} C_VEL
LIN {X 0,Y 417.474,Z 506.051,A -85,B 0,C 180,E1 -9987.106,E2 -9987.106} C_VEL
LIN {X 0,Y 417.644,Z 501.377,A -85,B 0,C 180,E1 -9988.554,E2 -9988.554} C_VEL
LIN {X 0,Y 418.2,Z 494.339,A -85,B 0,C 180,E1 -9990.241,E2 -9990.241} C_VEL
LIN {X 0,Y 418.662,Z 486.721,A -85,B 0,C 180,E1 -9991.684,E2 -9991.684} C_VEL
LIN {X 0,Y 419.313,Z 477.163,A -85,B 0,C 180,E1 -9993.123,E2 -9993.123} C_VEL
LIN {X 0,Y 419.911,Z 467.322,A -85,B 0,C 180,E1 -9994.32,E2 -9994.32} C_VEL
LIN {X 0,Y 420.59,Z 456.203,A -85,B 0,C 180,E1 -9995.394,E2 -9995.394} C_VEL
LIN {X 0,Y 421.276,Z 445.304,A -85,B 0,C 180,E1 -9996.226,E2 -9996.226} C_VEL
LIN {X 0,Y 421.657,Z 433.336,A -85,B 0,C 180,E1 -9996.941,E2 -9996.941} C_VEL
LIN {X 0,Y 422.085,Z 420.873,A -85,B 0,C 180,E1 -9997.475,E2 -9997.475} C_VEL
LIN {X 0,Y 422.435,Z 407.817,A -85,B 0,C 180,E1 -9997.829,E2 -9997.829} C_VEL
LIN {X 0,Y 423.432,Z 322.764,A -85,B 0,C 180,E1 -9999.274,E2 -9999.274} C_VEL
LIN {X 0,Y 419.81,Z 303.684,A -85,B 0,C 180,E1 -9999.766,E2 -9999.766} C_VEL
LIN {X 0,Y 419.087,Z 297.547,A -85,B 0,C 180,E1 -10001.12,E2 -10001.12} C_VEL
LIN {X 0,Y 418.397,Z 293.369,A -85,B 0,C 180,E1 -10002.09,E2 -10002.09} C_VEL
LIN {X 0,Y 418.305,Z 293.374,A -85,B 0,C 180,E1 -10005.595,E2 -10005.595} C_VEL
LIN {X 0,Y 418.28,Z 293.384,A -85,B 0,C 180,E1 -10008.618,E2 -10008.618} C_VEL
LIN {X 0,Y 418.239,Z 293.383,A -85,B 0,C 180,E1 -10011.697,E2 -10011.697} C_VEL
LIN {X 0,Y 418.249,Z 293.389,A -85,B 0,C 180,E1 -10014.853,E2 -10014.853} C_VEL
LIN {X 0,Y 418.211,Z 293.386,A -85,B 0,C 180,E1 -10018.07,E2 -10018.07} C_VEL
LIN {X 0,Y 418.243,Z 293.39,A -85,B 0,C 180,E1 -10021.019,E2 -10021.019} C_VEL
LIN {X 0,Y 418.238,Z 293.384,A -85,B 0,C 180,E1 -10023.679,E2 -10023.679} C_VEL
LIN {X 0,Y 418.243,Z 293.389,A -85,B 0,C 180,E1 -10027.225,E2 -10027.225} C_VEL
LIN {X 0,Y 418.212,Z 293.389,A -85,B 0,C 180,E1 -10030.867,E2 -10030.867} C_VEL
LIN {X 0,Y 418.208,Z 293.389,A -85,B 0,C 180,E1 -10033.728,E2 -10033.728} C_VEL
LIN {X 0,Y 418.205,Z 293.387,A -85,B 0,C 180,E1 -10036.447,E2 -10036.447} C_VEL
LIN {X 0,Y 418.211,Z 293.39,A -85,B 0,C 180,E1 -10039.133,E2 -10039.133} C_VEL
LIN {X 0,Y 418.24,Z 293.383,A -85,B 0,C 180,E1 -10042.775,E2 -10042.775} C_VEL
LIN {X 0,Y 418.238,Z 293.383,A -85,B 0,C 180,E1 -10046.321,E2 -10046.321} C_VEL
LIN {X 0,Y 418.247,Z 293.388,A -85,B 0,C 180,E1 -10049.728,E2 -10049.728} C_VEL
LIN {X 0,Y 418.231,Z 293.384,A -85,B 0,C 180,E1 -10053.018,E2 -10053.018} C_VEL
LIN {X 0,Y 418.261,Z 293.382,A -85,B 0,C 180,E1 -10056.217,E2 -10056.217} C_VEL
LIN {X 0,Y 418.255,Z 293.383,A -85,B 0,C 180,E1 -10059.337,E2 -10059.337} C_VEL
LIN {X 0,Y 418.283,Z 293.379,A -85,B 0,C 180,E1 -10062.396,E2 -10062.396} C_VEL
LIN {X 0,Y 418.305,Z 293.376,A -85,B 0,C 180,E1 -10065.403,E2 -10065.403} C_VEL
LIN {X 0,Y 418.308,Z 293.378,A -85,B 0,C 180,E1 -10068.368,E2 -10068.368} C_VEL
LIN {X 0,Y 418.451,Z 293.362,A -85,B 0,C 180,E1 -10072.278,E2 -10072.278} C_VEL
LIN {X 0,Y 418.488,Z 293.359,A -85,B 0,C 180,E1 -10074.217,E2 -10074.217} C_VEL
LIN {X 0,Y 418.538,Z 293.351,A -85,B 0,C 180,E1 -10078.075,E2 -10078.075} C_VEL
LIN {X 0,Y 418.455,Z 293.357,A -85,B 0,C 180,E1 -10080.962,E2 -10080.962} C_VEL
LIN {X 0,Y 418.472,Z 293.355,A -85,B 0,C 180,E1 -10082.888,E2 -10082.888} C_VEL
LIN {X 0,Y 418.473,Z 293.354,A -85,B 0,C 180,E1 -10085.783,E2 -10085.783} C_VEL
LIN {X 0,Y 418.37,Z 293.371,A -85,B 0,C 180,E1 -10088.696,E2 -10088.696} C_VEL
LIN {X 0,Y 418.358,Z 293.375,A -85,B 0,C 180,E1 -10092.614,E2 -10092.614} C_VEL
LIN {X 0,Y 418.295,Z 293.376,A -85,B 0,C 180,E1 -10095.594,E2 -10095.594} C_VEL
LIN {X 0,Y 418.278,Z 293.385,A -85,B 0,C 180,E1 -10098.617,E2 -10098.617} C_VEL
LIN {X 0,Y 418.237,Z 293.383,A -85,B 0,C 180,E1 -10101.696,E2 -10101.696} C_VEL
LIN {X 0,Y 418.247,Z 293.389,A -85,B 0,C 180,E1 -10104.852,E2 -10104.852} C_VEL
LIN {X 0,Y 418.209,Z 293.387,A -85,B 0,C 180,E1 -10108.069,E2 -10108.069} C_VEL
LIN {X 0,Y 418.24,Z 293.39,A -85,B 0,C 180,E1 -10111.019,E2 -10111.019} C_VEL
LIN {X 0,Y 418.235,Z 293.384,A -85,B 0,C 180,E1 -10113.678,E2 -10113.678} C_VEL
LIN {X 0,Y 418.241,Z 293.389,A -85,B 0,C 180,E1 -10117.224,E2 -10117.224} C_VEL
LIN {X 0,Y 418.209,Z 293.39,A -85,B 0,C 180,E1 -10120.867,E2 -10120.867} C_VEL
LIN {X 0,Y 418.205,Z 293.389,A -85,B 0,C 180,E1 -10123.728,E2 -10123.728} C_VEL
LIN {X 0,Y 418.202,Z 293.387,A -85,B 0,C 180,E1 -10126.447,E2 -10126.447} C_VEL
LIN {X 0,Y 418.209,Z 293.391,A -85,B 0,C 180,E1 -10129.133,E2 -10129.133} C_VEL
LIN {X 0,Y 418.237,Z 293.384,A -85,B 0,C 180,E1 -10132.775,E2 -10132.775} C_VEL
LIN {X 0,Y 418.235,Z 293.383,A -85,B 0,C 180,E1 -10136.321,E2 -10136.321} C_VEL
LIN {X 0,Y 418.245,Z 293.389,A -85,B 0,C 180,E1 -10139.727,E2 -10139.727} C_VEL
LIN {X 0,Y 418.31,Z 293.507,A -85,B 0,C 180,E1 -10142.304,E2 -10142.304} C_VEL
LIN {X 0,Y 420.958,Z 307.319,A -85,B 0,C 180,E1 -10145.105,E2 -10145.105} C_VEL
LIN {X 0,Y 420.722,Z 316.008,A -85,B 0,C 180,E1 -10146.745,E2 -10146.745} C_VEL
LIN {X 0,Y 419.614,Z 335.864,A -85,B 0,C 180,E1 -10150.428,E2 -10150.428} C_VEL
LIN {X 0,Y 419.317,Z 340.281,A -85,B 0,C 180,E1 -10151.24,E2 -10151.24} C_VEL
LIN {X 0,Y 423.119,Z 367.737,A -85,B 0,C 180,E1 -10151.868,E2 -10151.868} C_VEL
LIN {X 0,Y 422.214,Z 449.752,A -85,B 0,C 180,E1 -10153.282,E2 -10153.282} C_VEL
LIN {X 0,Y 421.628,Z 463.579,A -85,B 0,C 180,E1 -10153.725,E2 -10153.725} C_VEL
LIN {X 0,Y 421.099,Z 476.009,A -85,B 0,C 180,E1 -10154.325,E2 -10154.325} C_VEL
LIN {X 0,Y 420.365,Z 487.909,A -85,B 0,C 180,E1 -10155.104,E2 -10155.104} C_VEL
LIN {X 0,Y 419.812,Z 498.597,A -85,B 0,C 180,E1 -10156,E2 -10156} C_VEL
LIN {X 0,Y 419.088,Z 509.701,A -85,B 0,C 180,E1 -10157.161,E2 -10157.161} C_VEL
LIN {X 0,Y 418.466,Z 518.966,A -85,B 0,C 180,E1 -10158.373,E2 -10158.373} C_VEL
LIN {X 0,Y 417.852,Z 527.979,A -85,B 0,C 180,E1 -10159.827,E2 -10159.827} C_VEL
LIN {X 0,Y 417.503,Z 535.234,A -85,B 0,C 180,E1 -10161.285,E2 -10161.285} C_VEL
LIN {X 0,Y 417.259,Z 541.012,A -85,B 0,C 180,E1 -10162.742,E2 -10162.742} C_VEL
LIN {X 0,Y 417.115,Z 545.555,A -85,B 0,C 180,E1 -10164.197,E2 -10164.197} C_VEL
LIN {X 0,Y 417.138,Z 547.952,A -85,B 0,C 180,E1 -10165.167,E2 -10165.167} C_VEL
LIN {X 0,Y 417.024,Z 549.904,A -85,B 0,C 180,E1 -10166.134,E2 -10166.134} C_VEL
LIN {X 0,Y 417.088,Z 551.443,A -85,B 0,C 180,E1 -10167.102,E2 -10167.102} C_VEL
LIN {X 0,Y 417.091,Z 552.521,A -85,B 0,C 180,E1 -10168.068,E2 -10168.068} C_VEL
LIN {X 0,Y 417.054,Z 553.483,A -85,B 0,C 180,E1 -10169.999,E2 -10169.999} C_VEL
LIN {X 0,Y 417.056,Z 553.381,A -85,B 0,C 180,E1 -10170.965,E2 -10170.965} C_VEL
LIN {X 0,Y 417.09,Z 552.847,A -85,B 0,C 180,E1 -10171.931,E2 -10171.931} C_VEL
LIN {X 0,Y 417.072,Z 551.911,A -85,B 0,C 180,E1 -10172.897,E2 -10172.897} C_VEL
LIN {X 0,Y 417.108,Z 548.842,A -85,B 0,C 180,E1 -10174.832,E2 -10174.832} C_VEL
LIN {X 0,Y 417.135,Z 545.448,A -85,B 0,C 180,E1 -10176.253,E2 -10176.253} C_VEL
LIN {X 0,Y 417.347,Z 540.808,A -85,B 0,C 180,E1 -10177.742,E2 -10177.742} C_VEL
LIN {X 0,Y 417.728,Z 533.927,A -85,B 0,C 180,E1 -10179.441,E2 -10179.441} C_VEL
